// TIA Portal project "CropOne_SixRack" (V15.1)

(* hardware
DEVICE "ET 200SP station_1"  ET 200SP-Station
   slot 0: "Rack_0"  Rack  6ES5 710-8MAx1
   slot 1: "PLC"  CPU 1512SP-1 PN  6ES7 512-1DK01-0AB0  V2.6
   slot 2: "DQ 8x24VDC/0.5A ST_1"  DQ 8x24VDC/0.5A ST  6ES7 132-6BF01-0BA0  V0.0
      slot 1: "DQ 8x24VDC/0.5A ST_1"  DQ 8x24VDC/0.5A ST
   slot 3: "DQ 8x24VDC/0.5A ST_2"  DQ 8x24VDC/0.5A ST  6ES7 132-6BF01-0BA0  V0.0
      slot 1: "DQ 8x24VDC/0.5A ST_2"  DQ 8x24VDC/0.5A ST
   slot 4: "DQ 8x24VDC/0.5A ST_3"  DQ 8x24VDC/0.5A ST  6ES7 132-6BF01-0BA0  V0.0
      slot 1: "DQ 8x24VDC/0.5A ST_3"  DQ 8x24VDC/0.5A ST
   slot 5: "DQ 8x24VDC/0.5A ST_4"  DQ 8x24VDC/0.5A ST  6ES7 132-6BF01-0BA0  V0.0
      slot 1: "DQ 8x24VDC/0.5A ST_4"  DQ 8x24VDC/0.5A ST
   slot 6: "DQ 8x24VDC/0.5A ST_5"  DQ 8x24VDC/0.5A ST  6ES7 132-6BF01-0BA0  V0.0
      slot 1: "DQ 8x24VDC/0.5A ST_5"  DQ 8x24VDC/0.5A ST
   slot 7: "AI 4xU/I 2-wire ST_1"  AI 4xU/I 2-wire ST  6ES7 134-6HD01-0BA1  V2.0
      slot 1: "AI 4xU/I 2-wire ST_1"  AI 4xU/I 2-wire ST
   slot 8: "AI 4xU/I 2-wire ST_2"  AI 4xU/I 2-wire ST  6ES7 134-6HD01-0BA1  V2.0
      slot 1: "AI 4xU/I 2-wire ST_2"  AI 4xU/I 2-wire ST
   slot 9: "AI 4xU/I 2-wire ST_3"  AI 4xU/I 2-wire ST  6ES7 134-6HD01-0BA1  V2.0
      slot 1: "AI 4xU/I 2-wire ST_3"  AI 4xU/I 2-wire ST
   slot 10: "AI 4xU/I 2-wire ST_4"  AI 4xU/I 2-wire ST  6ES7 134-6HD01-0BA1  V2.0
      slot 1: "AI 4xU/I 2-wire ST_4"  AI 4xU/I 2-wire ST
   slot 11: "AI 4xU/I 2-wire ST_5"  AI 4xU/I 2-wire ST  6ES7 134-6HD01-0BA1  V2.0
      slot 1: "AI 4xU/I 2-wire ST_5"  AI 4xU/I 2-wire ST
   slot 12: "Server module_1"  Server module  6ES7 193-6PA00-0AA0  V1.1
      slot 1: "Server module_1"  Server module
   slot 127: "BA 2xRJ45"  BA 2xRJ45  6ES7 193-6AR00-0AA0  V0.0
      slot 32769: "Port_1"  6ES7 193-6AR00-0AA0
      slot 32770: "Port_2"  6ES7 193-6AR00-0AA0
DEVICE "SCALANCE S-600"  SCALANCE S-Station
   slot 0: "Rack"  Rail
   slot 0: "Router"  SCALANCE S615  6GK5 615-0AA00-2AA2  V5.0
DEVICE "SINAMICS G_1"  Sinamics.Device
   slot 0: "	_0"  Rail  SinamicsG120PRackP
   slot 0: "RackPumpVFD_1"  G120P CU230P-2 PN  6SL3243-0BB30-1FA0  4.7.10
      slot 1: "PROFINET interface"  MDD-SinamicsG120-P
   slot 3: "PM240-2 IP20"  PM240-2 IP20  6SL3210-1PB17-4ULx  -
DEVICE "ET 200SP station_2"  ET 200SP-Station
   slot 0: "Rack_0"  Rack  6ES5 710-8MAx1
   slot 0: "IO_Room_2"  IM 155-6 PN ST  6ES7 155-6AU01-0BN0  V4.1
   slot 1: "DQ 8x24VDC/0.5A ST_1"  DQ 8x24VDC/0.5A ST  6ES7 132-6BF01-0BA0  V0.0
      slot 1: "DQ 8x24VDC/0.5A ST_1"  DQ 8x24VDC/0.5A ST
   slot 2: "DQ 8x24VDC/0.5A ST_2"  DQ 8x24VDC/0.5A ST  6ES7 132-6BF01-0BA0  V0.0
      slot 1: "DQ 8x24VDC/0.5A ST_2"  DQ 8x24VDC/0.5A ST
   slot 3: "DQ 8x24VDC/0.5A ST_3"  DQ 8x24VDC/0.5A ST  6ES7 132-6BF01-0BA0  V0.0
      slot 1: "DQ 8x24VDC/0.5A ST_3"  DQ 8x24VDC/0.5A ST
   slot 4: "DQ 8x24VDC/0.5A ST_4"  DQ 8x24VDC/0.5A ST  6ES7 132-6BF01-0BA0  V0.0
      slot 1: "DQ 8x24VDC/0.5A ST_4"  DQ 8x24VDC/0.5A ST
   slot 5: "DQ 8x24VDC/0.5A ST_5"  DQ 8x24VDC/0.5A ST  6ES7 132-6BF01-0BA0  V0.0
      slot 1: "DQ 8x24VDC/0.5A ST_5"  DQ 8x24VDC/0.5A ST
   slot 6: "DQ 8x24VDC/0.5A ST_6"  DQ 8x24VDC/0.5A ST  6ES7 132-6BF00-0BA0  V1.1
      slot 1: "DQ 8x24VDC/0.5A ST_6"  DQ 8x24VDC/0.5A ST
   slot 7: "AI 4xU/I 2-wire ST_1"  AI 4xU/I 2-wire ST  6ES7 134-6HD01-0BA1  V2.0
      slot 1: "AI 4xU/I 2-wire ST_1"  AI 4xU/I 2-wire ST
   slot 8: "AI 4xU/I 2-wire ST_2"  AI 4xU/I 2-wire ST  6ES7 134-6HD01-0BA1  V2.0
      slot 1: "AI 4xU/I 2-wire ST_2"  AI 4xU/I 2-wire ST
   slot 9: "AI 4xU/I 2-wire ST_3"  AI 4xU/I 2-wire ST  6ES7 134-6HD01-0BA1  V2.0
      slot 1: "AI 4xU/I 2-wire ST_3"  AI 4xU/I 2-wire ST
   slot 10: "AI 4xU/I 2-wire ST_4"  AI 4xU/I 2-wire ST  6ES7 134-6HD01-0BA1  V2.0
      slot 1: "AI 4xU/I 2-wire ST_4"  AI 4xU/I 2-wire ST
   slot 11: "AI 4xU/I 2-wire ST_5"  AI 4xU/I 2-wire ST  6ES7 134-6HD01-0BA1  V2.0
      slot 1: "AI 4xU/I 2-wire ST_5"  AI 4xU/I 2-wire ST
   slot 12: "Server module_1"  Server module  6ES7 193-6PA00-0AA0  V1.1
      slot 1: "Server module_1"  Server module
   slot 127: "BA 2xRJ45"  BA 2xRJ45  6ES7 193-6AR00-0AA0  V0.0
      slot 1: "Port_1"  X1 P1 R  6ES7 193-6AR00-0AA0  V0.0
      slot 2: "Port_2"  X1 P2 R  6ES7 193-6AR00-0AA0  V0.0
DEVICE "HVAC_Modbus_1"  Dummy PC
   slot 1: "PROFINET interface"  PN-IO
DEVICE "HVAC_Modbus_2"  Dummy PC
   slot 1: "PROFINET interface"  PN-IO
DEVICE "SINAMICS G_2"  Sinamics.Device
   slot 0: "	_0"  Rail  SinamicsG120PRackP
   slot 0: "RackPumpVFD_2"  G120P CU230P-2 PN  6SL3243-0BB30-1FA0  4.7.10
      slot 1: "PROFINET interface"  MDD-SinamicsG120-P
   slot 3: "PM240-2 IP20"  PM240-2 IP20  6SL3210-1PB17-4ULx  -
DEVICE "SINAMICS G_3"  Sinamics.Device
   slot 0: "	_0"  Rail  SinamicsG120PRackP
   slot 0: "RackPumpVFD_3"  G120P CU230P-2 PN  6SL3243-0BB30-1FA0  4.7.10
      slot 1: "PROFINET interface"  MDD-SinamicsG120-P
   slot 3: "PM240-2 IP20"  PM240-2 IP20  6SL3210-1PB17-4ULx  -
DEVICE "SINAMICS G_4"  Sinamics.Device
   slot 0: "	_0"  Rail  SinamicsG120PRackP
   slot 0: "RackPumpVFD_4"  G120P CU230P-2 PN  6SL3243-0BB30-1FA0  4.7.10
      slot 1: "PROFINET interface"  MDD-SinamicsG120-P
   slot 3: "PM240-2 IP20"  PM240-2 IP20  6SL3210-1PB17-4ULx  -
DEVICE "SINAMICS G_5"  Sinamics.Device
   slot 0: "	_0"  Rail  SinamicsG120PRackP
   slot 0: "RackPumpVFD_5"  G120P CU230P-2 PN  6SL3243-0BB30-1FA0  4.7.10
      slot 1: "PROFINET interface"  MDD-SinamicsG120-P
   slot 3: "PM240-2 IP20"  PM240-2 IP20  6SL3210-1PB17-4ULx  -
DEVICE "SINAMICS G_6"  Sinamics.Device
   slot 0: "	_0"  Rail  SinamicsG120PRackP
   slot 0: "RackPumpVFD_6"  G120P CU230P-2 PN  6SL3243-0BB30-1FA0  4.7.10
      slot 1: "PROFINET interface"  MDD-SinamicsG120-P
   slot 3: "PM240-2 IP20"  PM240-2 IP20  6SL3210-1PB17-4ULx  -
*)

// ===== PLC "PLC"  CPU 1512SP-1 PN =====

VAR_GLOBAL CONSTANT   // PLC tag table "Library Constants"
   "eSTATE_MANUAL" : Int := 2;   // State Machine enumeration
   "ePBLT_FLASHING_ENABLED" : Int := 4;   // HMI PB LT enumeration
   "eSTATE_RETRACTING" : Int := 5;   // State Machine enumeration
   "IoScaling.S7Analog.Ni100.rScaledMax" : Real := 250.0;
   "IoScaling.S7Analog.Ni100.Climate.rScaledMax" : Real := 250.0;
   "eSTEP_StoppingStart" : Int := 4000;   // State Machine enumeration
   "eSTEP_VerifyCenterComplete" : Int := 7999;   // State Machine enumeration
   "IoScaling.S7Analog.150Ohms.rScaledMax" : Real := 150.0;
   "IoScaling.S7Analog.Default.bSwapBytes" : Bool := false;
   "eANALOG_INPUTHIGHHIGH" : Int := 102;
   "eMOTION_DISABLED" : Int := 4;   // Status Enumeration - Motion
   "IoScaling.S7Analog.Pt100.iRawMax" : Int := 8500;
   "eSTEP_RetractingComplete" : Int := 5999;   // State Machine enumeration
   "eMODE_MANUAL" : Int := 2;   // Mode enumeration
   "eANALOG_INPUTINVALID" : Int := 101;
   "ePBLT_HIDDEN" : Int := -1;   // HMI PB LT enumeration
   "eVALVE_HOMEON" : Int := 6;
   "IoScaling.S7Analog.Pt100.Climate.rScaledMin" : Real := -120.0;
   "eHOME_ABS_RET_ABS" : Int := 7;   // See MC_Home help for details
   "eMOTION_ERROR" : Int := 0;   // Status Enumeration - Motion
   "ePB_MAINTAINED" : Int := 1;   // HMI PB Type enumeration
   "LKINCTRL_LENGTH_OF_PATHDATA_NAME" : Int := 10;
   "LKINCTRL_NO_OF_PATHDATA_ELEMENTS" : Int := 15;
   "IoScaling.S7Analog.Pt100.Climate.iRawMax" : Int := 13000;
   "eVALVE_ERROR" : Int := 2;
   "IoScaling.S7Analog.Types.Pt100.Climate" : Int := 3;
   "eMODE_INDEPENDENT" : Int := 10;   // Mode
   "IoScaling.S7Analog.600Ohms.rScaledMax" : Real := 600.0;
   "eMOTION_RUNNING" : Int := 2;   // Status Enumeration - Motion
   "IoScaling.S7Analog.Ni100.Climate.rScaledMin" : Real := -60.0;
   "eMOTION_STOPPED" : Int := 1;   // Status Enumeration - Motion
   "eMOTION_MAINTENANCE" : Int := 3;   // Status Enumeration - Motion
   "IoScaling.S7Analog.Ni100.rScaledMin" : Real := -60.0;
   "eSTATE_STOPPING" : Int := 4;   // State Machine enumeration
   "IoScaling.S7Analog.Pt100.Climate.rScaledMax" : Real := 130.0;
   "IoScaling.S7Analog.Pt100.rScaledMax" : Real := 850.0;
   "IoScaling.S7Analog.Types.Ni100.Climate" : Int := 5;
   "ePB_UNLATCH" : Int := 3;   // HMI PB Type enumeration
   "IoScaling.S7Analog.Ni100.Climate.iRawMax" : Int := 25000;
   "eSTEP_BladeChangeStart" : Int := 6000;   // State Machine enumeration
   "IoScaling.S7Analog.300Ohms.rScaledMin" : Real := 0.0;
   "IoScaling.S7Analog.Types.Pt100" : Int := 2;
   "LKINCTRL_PI" : LReal := 3.1415926535897932846264;
   "eVALVE_WORKPOSITION" : Int := 3;
   "eCAM_SYNCDIRECTION_SHORTESTWAY" : Int := 3;   // See MC_CamIn help for details
   "IoScaling.S7Analog.Types.+-V/mA" : Int := 1;
   "ePBLT_FLASHING_DISABLED" : Int := 5;   // HMI PB LT enumeration
   "IoScaling.S7Analog.150Ohms.rScaledMin" : Real := 0.0;
   "eHOME_ACCEPT_CURRENT" : Int := 11;   // Used when the configured and current encoders don't match
   "LKINCTRL_NO_OF_START_EXECUTE_CMDS" : Int := 5;
   "ePBLT_TRANSITIONING" : Int := 2;   // HMI PB LT enumeration
   "SM_ACTIVE_DYNAMICS" : Int := 0;
   "eVALVE_WORKON" : Int := 5;
   "IoScaling.S7Analog.+-V/mA.iRawMax" : Int := 27648;
   "eSTATE_INITIALIZATION" : Int := 1;   // State Machine enumeration
   "LKINCTRL_NO_OF_PATHDATA_PREBUFFER_ELEMENTS" : Int := 5;
   "eHOME_ABS_RET_OFFSET" : Int := 6;   // See MC_Home help for details
   "eSTEP_BladeChangeComplete" : Int := 6999;   // State Machine enumeration
   "eSTEP_RunningComplete" : Int := 3999;   // State Machine enumeration
   "eANALOG_READY" : Int := 100;
   "ePBLT_ENABLED" : Int := 1;   // HMI PB LT enumeration
   "IoScaling.S7Analog.Pt100.Climate.iRawMin" : Int := -12000;
   "eSTATE_RUNNING" : Int := 3;   // State Machine enumeration
   "LKINCTRL_NO_OF_LAST_FLAG" : Int := 15;
   "IoScaling.S7Analog.Ni100.iRawMax" : Int := 2500;
   "IoScaling.S7Analog.Types.Default" : Int := 0;
   "eHOME_ACCEPT_CONFIG" : Int := 12;   // Used when the configured and current encoders don't match
   "eSTEP_RunningStart" : Int := 3000;   // State Machine enumeration
   "IoScaling.S7Analog.Default.iRawMin" : Int := 0;
   "ePBLT_ACTIVE" : Int := 3;   // HMI PB LT enumeration
   "IoScaling.S7Analog.Types.Ni100" : Int := 4;
   "eMODE_AUTO" : Int := 1;   // Mode enumeration
   "IoScaling.S7Analog.Default.iRawMax" : Int := 27648;
   "ePBLT_DISABLED" : Int := 0;   // HMI PB LT enumeration
   "LKINCTRL_NO_OF_SEQ_EXECUTE_CMDS" : Int := 5;
   "eSTEP_StoppingComplete" : Int := 4999;   // State Machine enumeration
   "IoScaling.S7Analog.Ni100.Climate.iRawMin" : Int := -6000;
   "IoScaling.S7Analog.Pt100.iRawMin" : Int := -2000;
   "ePB_LATCH" : Int := 2;   // HMI PB Type enumeration
   "eVALVE_ESTOP" : Int := 1;
   "eSTEP_RetractingStart" : Int := 5000;   // State Machine enumeration
   "IoScaling.S7Analog.300Ohms.rScaledMax" : Real := 300.0;
   "eANALOG_INPUTLOW" : Int := 105;
   "IoScaling.S7Analog.Pt100.rScaledMin" : Real := -200.0;
   "eSTATE_BLADECHANGE" : Int := 6;   // State Machine enumeration
   "IoScaling.S7Analog.600Ohms.rScaledMin" : Real := 0.0;
   "eSTATE_VERIFYCENTER" : Int := 7;   // State Machine enumeration
   "eVALVE_STOPPED" : Int := 0;
   "eCAM_SYNCPROFILEREFERENCE_LEADINGVALUEDISTANCE" : Int := 1;   // See MC_CamIn help for details
   "IoScaling.S7Analog.Ni100.iRawMin" : Int := -600;
   "ePB_HELD" : Int := 4;   // HMI PB Type enumeration
   "LKINCTRL_NO_OF_CMD_SETFLAGS" : Int := 8;
   "eSTEP_VerifyCenterStart" : Int := 7000;   // State Machine enumeration
   "eVALVE_HOMEPOSITION" : Int := 4;
   "eANALOG_INPUTHIGH" : Int := 104;
   "eANALOG_INPUTLOWLOW" : Int := 103;
   "IoScaling.S7Analog.+-V/mA.iRawMin" : Int := -27648;
   "ePB_MOMENTARY" : Int := 0;   // HMI PB Type enumeration
   "Modes.PID.Pretuning" : Int := 1;
   "TotalizerTimeUnits.DAYS" : Int := 4;
   "HMI.Status.ForwardWork" : Int := 3;
   "FIFO.iQueueDisabled" : Int := -1;
   "Handshakes.iSize" : Int := 5;
   "Modes.Auto" : Int := 1;
   "HMI.Status.Generic1" : Int := 101;
   "Simocode.Types.DirectStarter" : Int := 1;
   "Estop.MinSetPoint" : Int := 0;
   "Simocode.Types.OverloadRelay" : Int := 0;
   "HMI.Status.SimulatedReverseHome" : Int := 8;
   "TotalizerTimeUnits.MILLISECONDS" : Int := 0;
   "HMI.Status.Generic4" : Int := 104;
   "SoftStarter.HMI.Status.EStop" : Int := 1;
   "HMI.Status.OnForwardWork" : Int := 5;
   "DataTypes.iMaxInt" : Int := 32767;
   "FIFO.iQueueSize" : Int := 5;
   "Modes.PID.ManualMode" : Int := 4;
   "TotalizerTimeUnits.SECONDS" : Int := 1;
   "SoftStarter.Types.3RW30" : Int := 30;
   "HMI.Status.Generic3" : Int := 103;
   "HMI.Status.OnReverseHome" : Int := 6;
   "HMI.Status.Estop" : Int := 1;
   "SoftStarter.HMI.Status.Error" : Int := 2;
   "HMI.Status.Generic6" : Int := 106;
   "DataTypes.rMaxReal" : Real := 3.402823e38;
   "SoftStarter.HMI.Status.Off" : Int := 0;
   "Modes.PID.Inactive" : Int := 0;
   "HMI.Status.GenericNone" : Int := 100;
   "HMI.Status.Generic2" : Int := 102;
   "Modes.PID.AutoMode" : Int := 3;
   "SoftStarter.HMI.Status.On" : Int := 4;
   "Estop.HMISetPoint" : Int := 2;
   "HMI.Status.ReverseHome" : Int := 4;
   "DataTypes.rMinReal" : Real := -3.402823e38;
   "TotalizerTimeUnits.MINUTES" : Int := 2;
   "Modes.PID.FineTuning" : Int := 2;
   "TotalizerTimeUnits.HOURS" : Int := 3;
   "Ramp.Timed" : Int := 1;
   "Estop.MaxSetPoint" : Int := 1;
   "SoftStarter.Types.3RW40" : Int := 40;
   "Ramp.Continuous" : Int := 0;
   "HMI.Status.Generic5" : Int := 105;
   "Modes.Manual" : Int := 2;
   "Modes.Stop" : Int := 0;
   "HMI.Status.SimulatedOnReverseHome" : Int := 10;
   "Simocode.Types.ReversingStarter" : Int := 2;
   "Modes.Independent" : Int := 10;
   "DataTypes.iMinInt" : Int := -32768;
   "SoftStarter.HMI.Status.RampUp" : Int := 3;
   "SoftStarter.HMI.Status.RampDown" : Int := 5;
   "HMI.Status.Error" : Int := 2;
   "HMI.Status.SimulatedOnForwardWork" : Int := 9;
   "HMI.Status.SimulatedForwardWork" : Int := 7;
   "HMI.Status.Stopped" : Int := 0;
END_VAR

VAR_GLOBAL   // PLC tag table "IO"
   "GlobalAI" AT %I100.0 : "udtArrAIGlobal";
   "GlobalDQ" AT %Q100.0 : "udtArrDQGlobal";
END_VAR

VAR_GLOBAL CONSTANT   // PLC tag table "GLOBAL_CONSTANTS"
   "NUM_AI_RACK" : UInt := 1;   // Number of physical analog input points used per rack.
   "NUM_DQ_RACK" : UInt := 4;   // Number of physical digital output points used per rack.
   "NUM_DQ_ROOM" : UInt := 8;   // Number of physical digital output points used per room.
   "MAX_DQ_PER_ROOM" : UInt := 40;   // Max number of physical digital output points per room-based IO module. This needs to equal (NUM_DQ_ROOM + NUM_DQ_RACK*MAX_RACKS_PER_ROOM + EXTRA_DQ_PER_ROOM).
   "MAX_VFDS" : UInt := 6;   // Total number of VFDs configured in the HW config. This needs to equal MAX_ROOMS * MAX_RACKS_PER_ROOM.
   "MAX_ROOMS" : UInt := 1;   // Maximum possible number of rooms controlled by a given PLC
   "MAX_RACKS_PER_ROOM" : UInt := 6;   // Maximum possible number of racks per room
   "NUM_AI_ROOM" : UInt := 12;   // Number of physical analog input points used per room.
   "EXTRA_DQ_PER_ROOM" : UInt := 8;   // Number of unused physical digital output points per room-based IO module.
   "EXTRA_AI_PER_ROOM" : UInt := 2;   // Number of unused physical analog input points per room-based IO module.
   "MAX_AI_PER_ROOM" : UInt := 20;   // Max number of physical analog input points per room-based IO module. This needs to equal (NUM_AI_ROOM + NUM_AI_RACK*MAX_RACKS_PER_ROOM + EXTRA_AI_PER_ROOM).
END_VAR

VAR_GLOBAL   // PLC tag table "System Bits"
   "System_Byte" AT %MB1 : Byte;
   "AlwaysFALSE" AT %M1.3 : Bool;
   "Clock_1.25Hz" AT %M0.4 : Bool;
   "Clock_1Hz" AT %M0.5 : Bool;
   "Clock_0.5Hz" AT %M0.7 : Bool;
   "FirstScan" AT %M1.0 : Bool;
   "Clock_Byte" AT %MB0 : Byte;
   "Clock_2.5Hz" AT %M0.2 : Bool;
   "Clock_0.625Hz" AT %M0.6 : Bool;
   "Clock_5Hz" AT %M0.1 : Bool;
   "Clock_10Hz" AT %M0.0 : Bool;
   "AlwaysTRUE" AT %M1.2 : Bool;
   "DiagStatusUpdate" AT %M1.1 : Bool;
   "Clock_2Hz" AT %M0.3 : Bool;
END_VAR

VAR_GLOBAL   // PLC tag table "Temporary I/O"
   "Q_DischargeSolenoid" AT %Q0.2 : Bool;
   "Q_Rack3Supply" AT %Q1.5 : Bool;
   "Q_Rack4Lights" AT %Q3.4 : Bool;
   "IW_pHSensor" AT %IW12 : Int;
   "IW_RoomTemperature_1" AT %IW0 : Int;
   "Q_Rack6Supply" AT %Q2.6 : Bool;
   "Q_Rack5Lights" AT %Q3.5 : Bool;
   "Q_Rack4Supply" AT %Q2.0 : Bool;
   "Q_Rack1Return" AT %Q1.0 : Bool;
   "Q_Rack2Lights" AT %Q3.2 : Bool;
   "IW_NutrientALevel" AT %IW6 : Int;
   "Q_Rack3Lights" AT %Q3.3 : Bool;
   "Q_Rack2Shelves" AT %Q1.4 : Bool;
   "Q_FreshWaterSolenoid" AT %Q0.1 : Bool;
   "IW_Rack4Level" AT %IW24 : Int;
   "Q_MPathSolenoid" AT %Q0.0 : Bool;
   "Q_Rack4Shelves" AT %Q2.2 : Bool;
   "Q_Rack5Supply" AT %Q2.3 : Bool;
   "Q_NutrientAEnable" AT %Q0.4 : Bool;
   "IW_TankLevel" AT %IW4 : Int;
   "Q_Rack1Lights" AT %Q3.1 : Bool;
   "Q_Rack4Return" AT %Q2.1 : Bool;
   "Q_Rack6Lights" AT %Q3.6 : Bool;
   "IW_ISESensor" AT %IW16 : Int;
   "Q_Rack3Return" AT %Q1.6 : Bool;
   "Q_Rack6Shelves" AT %Q3.0 : Bool;
   "IW_NutrientAcidLevel" AT %IW10 : Int;
   "Q_Rack1Supply" AT %Q0.7 : Bool;
   "Q_NutrientMixingPumps" AT %Q3.7 : Bool;
   "Q_NutrientBEnable" AT %Q0.5 : Bool;
   "Q_Rack5Return" AT %Q2.4 : Bool;
   "Q_NutrientAcidEnable" AT %Q0.6 : Bool;
   "Q_Rack3Shelves" AT %Q1.7 : Bool;
   "Q_Rack2Return" AT %Q1.3 : Bool;
   "Q_Rack5Shelves" AT %Q2.5 : Bool;
   "IW_Rack2Level" AT %IW20 : Int;
   "IW_Rack6Level" AT %IW28 : Int;
   "IW_NutrientBLevel" AT %IW8 : Int;
   "Q_Rack1Shelves" AT %Q1.1 : Bool;
   "Q_Rack2Supply" AT %Q1.2 : Bool;
   "IW_Rack1Level" AT %IW18 : Int;
   "IW_RoomHumidity_1" AT %IW2 : Int;
   "IW_Rack3Level" AT %IW22 : Int;
   "Q_TankReturnSolenoid" AT %Q0.3 : Bool;
   "IW_Rack5Level" AT %IW26 : Int;
   "Q_Rack6Return" AT %Q2.7 : Bool;
   "IW_ECSensor" AT %IW14 : Int;
   "IW_RoomTemperature_2" AT %IW32 : Int;
   "IW_RoomHumidity_2" AT %IW34 : Int;
   "IW_ORPSensor" AT %IW36 : Int;
END_VAR

TYPE "udtTimeOfDaySetpoint"
   STRUCT
      TimeOfDaySeconds : DInt := -1;   // -1 default for unused setpoint
      rSetpoint : Real;
   END_STRUCT;
END_TYPE

TYPE "udtModbusValReal"
   STRUCT
      iRegister : UInt;   // Full modbus address (1 indexed, including offset for object type)
      rVal : Real;
   END_STRUCT;
END_TYPE

TYPE "udtNutrientReading"
   STRUCT
      rISEReading : Real;   // Nutrient measurement level
      rORPReading : Real;   // Nutrient measurement level
      rECReading : Real;   // Nutrient measurement level
      rpHReading : Real;   // Nutrient measurement level
   END_STRUCT;
END_TYPE

TYPE "udtModbusValBool"
   STRUCT
      iAddr : UInt;   // Full modbus address (1 indexed, including offset for object type)
      bVal : Bool;
   END_STRUCT;
END_TYPE

TYPE "udtFertigationSettings"
   STRUCT
      tMeasurementTime : Time;   // Duration of cycle through M loop before measurement taken (s)
      rMeasurementVolume : Real;   // Amount of water to receive from rack for measurement (L)
      bNutrientAEnable : Bool;   // Enables nutrient A for use in dosing
      bNutrientBEnable : Bool;   // Enables nutrient B for use in dosing
      rISELowSP : Real;   // Low setpoint for ISE measurement for dosing
      rISEHighSP : Real;   // High setpoint for ISE measurement for dosing
      tNutrientDosingDuration : Time;   // Duration for which to add a nutrient during dosing (s)
      bDosingActive : Bool;   // Rack was dosed on last MD cycle and is below high SP
      rOperatingVolume : Real;   // Operating volume for fill after dosing (L)
      rTotalShelfVolume : Real;
      rMaxReservoirVolume : Real;   // Maximum water capacity of the rack (L)
      rRackCurrentVolume : Real;   // Current rack fill level (L)
      bPumpAtStandstill : Bool;
      bEndDischargeCommand : Bool;
      tDischargeTime : Time;
      bEnableIncomingRotate : Bool;   // Rack is in M&D mode and circulating state
   END_STRUCT;
END_TYPE

// folder: IO

TYPE "udtDigitalOutput"
   STRUCT
      bAutoVal : Bool;   // Value set by the program
      bOverrideVal : Bool;   // Value set by the user, tracks bAuto when bOverrideEnable=0
      bStatus : Bool;   // Value being written to actual output
      bOverrideEnable : Bool;   // Sets bOut to bOverride
   END_STRUCT;
END_TYPE

TYPE "udtArrDQRoom"
   STRUCT
      DQ : Array[1.."MAX_DQ_PER_ROOM"] of Bool;
   END_STRUCT;
END_TYPE

TYPE "udtArrAIRoom"
   STRUCT
      AI : Array[1.."MAX_AI_PER_ROOM"] of Int;
   END_STRUCT;
END_TYPE

TYPE "udtArrDQGlobal"
   STRUCT
      Room : Array[1.."MAX_ROOMS"] of "udtArrDQRoom";
   END_STRUCT;
END_TYPE

TYPE "udtArrAIGlobal"
   STRUCT
      Room : Array[1.."MAX_ROOMS"] of "udtArrAIRoom";
   END_STRUCT;
END_TYPE

TYPE "udtRackDQ"
   STRUCT
      Q_SupplySolenoid : Bool;
      Q_ReturnSolenoid : Bool;
      Q_ShelfSolenoid : Bool;
      Q_Lights : Bool;
   END_STRUCT;
END_TYPE

TYPE "udtRoomAI"
   STRUCT
      IW_RoomTemperature_1 : Int;
      IW_RoomTemperature_2 : Int;
      IW_RoomHumidity_1 : Int;
      IW_RoomHumidity_2 : Int;
      IW_TankLevel : Int;
      IW_NutrientALevel : Int;
      IW_NutrientBLevel : Int;
      IW_NutrientAcidLevel : Int;
      IW_pHSensor : Int;
      IW_ECSensor : Int;
      IW_ISESensor : Int;
      IW_ORPSensor : Int;
   END_STRUCT;
END_TYPE

TYPE "udtRoomDQ"
   STRUCT
      Q_MPathSolenoid : Bool;
      Q_FreshWaterSolenoid : Bool;
      Q_DischargeSolenoid : Bool;
      Q_TankReturnSolenoid : Bool;
      Q_NutrientAEnable : Bool;
      Q_NutrientBEnable : Bool;
      Q_NutrientAcidEnable : Bool;
      Q_NutrientMixingPumps : Bool;
   END_STRUCT;
END_TYPE

TYPE "udtRackAI"
   STRUCT
      IW_ReservoirLevel : Int;
   END_STRUCT;
END_TYPE

// folder: Library Data Types/Error

TYPE "udtError_VFD"
VERSION : 0.1
   STRUCT
      MotorProtectorTripped : Bool;   // Motor protector tripped
      LocalDisconnectOff : Bool;   // Motor disconnect off
      ClutchTripped : Bool;   // Clutch tripped
      NoContactorFeedback : Bool;   // No feedback from motor contactor
      ContactorStillOn : Bool;   // Contactor still on
      NoSignalForward : Bool;   // No signal forward from VFD
      NoSignalReverse : Bool;   // No signal reverse from VFD
      MotorNotStopped : Bool;   // Motor doesn't stop
      MaxFrequencyReached : Bool;   // Max frequency reached
      Overcurrent : Bool;   // VFD overcurrent
      MotorOverload : Bool;   // Motor overload
      VFDOverload : Bool;   // VFD overload
      GeneralFault : Bool;   // VFD fault
      NoCoolingFanFeedback : Bool;   // No feedback from cooling fan
   END_STRUCT;
END_TYPE

// folder: Library Data Types/HMI

TYPE "udtHMI_VFD_Control"
VERSION : 0.1
   STRUCT
      iMode : Int;   // Current mode
      iErrorCode : Int;   // Error code
      iStatus : Int;   // Status for HMI display
      rManualSpeedSP : Real;   // Speed set point for manual mode
      rAutoSpeedSP : Real;   // Speed set point for automatic mode
      rActualSpeed : Real;   // Actual motor speed
      rActualCurrent : Real;   // Actual motor current
      rActualPower : Real;   // Actual motor power
      bPB_ResetError : Bool;   // PB Reset errors
      bPB_Forward : Bool;   // PB Move forward in manual mode
      bPB_Reverse : Bool;   // PB Move reverse in manual mode
      bPB_Stop : Bool;   // PB Stop in manual mode
      bPBEN_ResetError : Bool;   // PB Reset errors enabled
      bPBEN_Forward : Bool;   // PB Forward enabled
      bPBEN_Reverse : Bool;   // PB Reverse enabled
      bPBEN_Stop : Bool;   // PB Stop enabled
      bForwardOn : Bool;   // Moving forward
      bReverseOn : Bool;   // Moving Reverse
      bSignalForward : Bool;   // Forward signal
      bSignalReverse : Bool;   // Reverse signal
      bError : Bool;   // Overall error
      bInterlock : Bool;   // VFD Interlocked
   END_STRUCT;
END_TYPE

// folder: (top level)

DATA_BLOCK "dbMain"   // DB6
{ S7_Optimized_Access := 'TRUE' }
VERSION : 0.1
// stored: InstanceOfName fbMain
"fbMain"
BEGIN
END_DATA_BLOCK

FUNCTION_BLOCK "fbRoomHVAC"   // FB2, LAD
{ S7_Optimized_Access := 'TRUE' }
VERSION : 0.1
   VAR
      Temperature_Cooling : "fbAlarmedSetpoint";
      Humidity : "fbAlarmedSetpoint";
      CO2 : "fbAlarmedSetpoint";
   END_VAR
   VAR RETAIN
      Controls : Struct
         rHeatingSP : Real := 55.0;
         bResetAlarm : Bool;
         bResetModbus : Bool;
      END_STRUCT;
   END_VAR
   VAR
      Status : Struct
         rSupplyAirTemperature : Real;
         bModbusError : Bool;
         wLastModbusErrorCode : Word;
         Compressor_1_Percentage : Real;
         Compressor_2_Percentage : Real;
         ZoneAirEnthalpy : Real;
         Compressor_1_Command : Bool;
         Compressor_1_Enabled : Bool;
         Compressor_1_Alarm : Bool;
         Compressor_2_Command : Bool;
         Compressor_2_Enabled : Bool;
         Compressor_2_Alarm : Bool;
         LPS1_Alarm : Bool;
         LPS2_Alarm : Bool;
         HPS1_Alarm : Bool;
         HPS2_Alarm : Bool;
      END_STRUCT;
   END_VAR
   VAR RETAIN
      Config : Struct
         ModbusServerAddr : IP_V4;   // IP address for Modbus TCP server
         ID : UInt := 81;   // Unique ID for connection, also used as port number on PLC
      END_STRUCT;
   END_VAR
   VAR
      TCPConnection : TCON_IP_v4;
      fbModbusTCPClient_Instance : "fbModbusTCPClient";
      Read_Discrete : Array[0..9] of "udtModbusValBool";
      Write_Discrete : Array[0..0] of "udtModbusValBool";
      Read_Registers : Array[0..6] of "udtModbusValReal";
      Write_Registers : Array[0..2] of "udtModbusValReal";
   END_VAR
   VAR CONSTANT
      cFakeScaling : Int := 150;
      cRoomTempIndex : Int := 0;
      cHumidityIndex : Int := 1;
      cCO2Index : Int := 2;
      cSupplyAirTempIndex : Int := 3;
   END_VAR
   // TCPConnection.RemotePort := 502;
   // TCPConnection.ActiveEstablished := true;
   // TCPConnection.ConnectionType := 11;
   // Config.ModbusServerAddr.ADDR[2] := 1;
   // Config.ModbusServerAddr.ADDR[1] := 10;
   // TCPConnection.LocalPort := 1001;
   // TCPConnection.RemoteAddress.ADDR[1] := 10;
   // TCPConnection.RemoteAddress.ADDR[2] := 1;
   // TCPConnection.RemoteAddress.ADDR[3] := 0;
   // TCPConnection.RemoteAddress.ADDR[4] := 20;
   // Config.ModbusServerAddr.ADDR[3] := 0;
   // Config.ModbusServerAddr.ADDR[4] := 20;
   // Temperature_Cooling.arrSetpoints[1].rSetpoint := 75.0;
   // Humidity.arrSetpoints[1].rSetpoint := 55.0;
BEGIN

REGION Network 1 (SCL): Set connection parameters
   #TCPConnection.InterfaceId := "Local~PROFINET_interface_1"; // PLC ethernet port
   #TCPConnection.ID := UINT_TO_WORD(#Config.ID);
   #TCPConnection.ConnectionType := 11; // TCP
   #TCPConnection.ActiveEstablished := TRUE;
   #TCPConnection.RemoteAddress := #Config.ModbusServerAddr;
   #TCPConnection.RemotePort := 502; // Default for Modbus TCP
   #TCPConnection.LocalPort := #Config.ID;
END_REGION

REGION Network 2 (SCL): Set up registers
   // Read coils and discrete inputs (00001 and 10001)
   #Read_Discrete[0].iAddr := 10048; // Compressor_1_Command
   #Read_Discrete[1].iAddr := 10067; // Compressor_1_Enabled
   #Read_Discrete[2].iAddr := 10091; // Compressor_1_Alarm
   #Read_Discrete[3].iAddr := 10049; // Compressor_2_Command
   #Read_Discrete[4].iAddr := 10008; // Compressor_2_Enabled
   #Read_Discrete[5].iAddr := 10068; // Compressor_2_Alarm
   #Read_Discrete[6].iAddr := 10089; // LPS1_Alarm
   #Read_Discrete[7].iAddr := 10034; // LPS2_Alarm
   #Read_Discrete[8].iAddr := 10093; // HPS1_Alarm
   #Read_Discrete[9].iAddr := 10097; // HPS2_Alarm

   // Write coils (00001)
   #Write_Discrete[0].iAddr := 00020; // Alarm reset
   #Write_Discrete[0].bVal := #Controls.bResetAlarm;

   // Read input and holding registers (30001 and 40001)
   #Read_Registers[#cRoomTempIndex].iRegister      := 30035; // Room Temperature
   #Read_Registers[#cHumidityIndex].iRegister      := 30031; // Humidity
   #Read_Registers[#cCO2Index].iRegister           := 30001; // CO2
   #Read_Registers[#cSupplyAirTempIndex].iRegister := 30043; // Supply Air Temperature

   #Read_Registers[4].iRegister := 30077; // Compressor_1_percentage
   #Read_Registers[5].iRegister := 30049; // Compressor_2_percentage
   #Read_Registers[6].iRegister := 30039; // ZoneAirEnthalpy

   // Write holding registers (40001)
   #Write_Registers[0].iRegister := 40119; // Cooling SP
   #Write_Registers[0].rVal := #Temperature_Cooling.rSetpoint;

   #Write_Registers[1].iRegister := 40121; // Heating SP
   #Write_Registers[1].rVal := #Controls.rHeatingSP;

   #Write_Registers[2].iRegister := 40097; // Dehumidification SP
   #Write_Registers[2].rVal := #Humidity.rSetpoint;
   (*
   #Write_Data[3].iRegister := 2; // CO2 SP 1
   #Write_Data[3].rVal := #CO2.rSetpoint;

   #Write_Data[4].iRegister := 66; // CO2 SP 2
   #Write_Data[4].rVal := #CO2.rSetpoint;
   *)
END_REGION

REGION Network 3: Modbus TCP Client Block Call
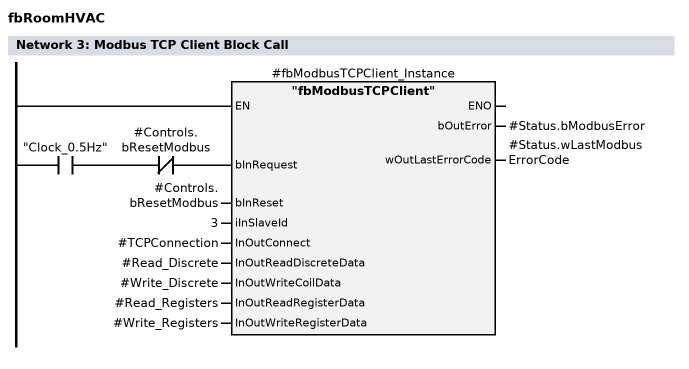
   RUNG wire#powerrail
      #fbModbusTCPClient_Instance(bInRequest := wire#w1, bInReset := #Controls.bResetModbus, iInSlaveId := 3, InOutConnect := #TCPConnection, InOutReadDiscreteData := #Read_Discrete, InOutWriteCoilData := #Write_Discrete, InOutReadRegisterData := #Read_Registers, InOutWriteRegisterData := #Write_Registers, bOutError => #Status.bModbusError, wOutLastErrorCode => #Status.wLastModbusErrorCode)
   END_RUNG
   RUNG wire#powerrail
      Contact( "Clock_0.5Hz" )
      I_Contact( #Controls.bResetModbus )
   END_RUNG wire#w1
   // the same network as SCL:
   #fbModbusTCPClient_Instance(bInRequest := "Clock_0.5Hz" AND NOT #Controls.bResetModbus,   // "fbModbusTCPClient"
                           bInReset := #Controls.bResetModbus,
                           iInSlaveId := 3,
                           InOutConnect := #TCPConnection,
                           InOutReadDiscreteData := #Read_Discrete,
                           InOutWriteCoilData := #Write_Discrete,
                           InOutReadRegisterData := #Read_Registers,
                           InOutWriteRegisterData := #Write_Registers,
                           bOutError => #Status.bModbusError,
                           wOutLastErrorCode => #Status.wLastModbusErrorCode);
END_REGION

REGION Network 4 (SCL): Parse received data
   // Status data
   #Status.Compressor_1_Percentage := #Read_Registers[4].rVal;
   #Status.Compressor_2_Percentage := #Read_Registers[5].rVal;
   #Status.ZoneAirEnthalpy := #Read_Registers[6].rVal;

   #Status.Compressor_1_Command := #Read_Discrete[0].bVal;
   #Status.Compressor_1_Enabled := #Read_Discrete[1].bVal;
   #Status.Compressor_1_Alarm :=   #Read_Discrete[2].bVal;
   #Status.Compressor_2_Command := #Read_Discrete[3].bVal;
   #Status.Compressor_2_Enabled := #Read_Discrete[4].bVal;
   #Status.Compressor_2_Alarm :=   #Read_Discrete[5].bVal;
   #Status.LPS1_Alarm := #Read_Discrete[6].bVal;
   #Status.LPS2_Alarm := #Read_Discrete[7].bVal;
   #Status.HPS1_Alarm := #Read_Discrete[8].bVal;
   #Status.HPS2_Alarm := #Read_Discrete[9].bVal;


   // Bypass analog scaling for alarmed setpoints
   #Temperature_Cooling.Config.rLowCalibration := 0;
   #Temperature_Cooling.Config.rHighCalibration := #cFakeScaling;
   #Humidity.Config.rLowCalibration := 0;
   #Humidity.Config.rHighCalibration := #cFakeScaling;
   #CO2.Config.rLowCalibration := 0;
   #CO2.Config.rHighCalibration := #cFakeScaling;

   #Temperature_Cooling(
                        iInRawValue := REAL_TO_INT(#Read_Registers[#cRoomTempIndex].rVal /
                                                   #cFakeScaling * "IoScaling.S7Analog.Default.iRawMax"));

   #Humidity(
             iInRawValue := REAL_TO_INT(#Read_Registers[#cHumidityIndex].rVal /
                                        #cFakeScaling * "IoScaling.S7Analog.Default.iRawMax"));

   #CO2(
        iInRawValue := REAL_TO_INT(#Read_Registers[#cCO2Index].rVal /
                                   #cFakeScaling * "IoScaling.S7Analog.Default.iRawMax"));

   #Status.rSupplyAirTemperature := #Read_Registers[#cSupplyAirTempIndex].rVal;
END_REGION
END_FUNCTION_BLOCK

FUNCTION_BLOCK "fbRoom"   // FB3, LAD
{ S7_Optimized_Access := 'TRUE' }
VERSION : 0.1
   VAR_INPUT
      arrAI : Array[1.."NUM_AI_ROOM"] of Int;
      AI AT arrAI : "udtRoomAI";
   END_VAR
   VAR_OUTPUT
      arrDQ : Array[1.."NUM_DQ_ROOM"] of Bool;
      DQ AT arrDQ : "udtRoomDQ";
   END_VAR
   VAR
      Rack : Array[1.."MAX_RACKS_PER_ROOM"] of "fbRack";
      Fertigation : "fbRoomFertigation";
      HVAC : "fbRoomHVAC";
   END_VAR
   VAR RETAIN
      Config : Struct
         iNumRacks : Int := 1;
      END_STRUCT;
   END_VAR
   VAR
      AI_Temperature_1 : "fbAlarmedSetpoint";
      AI_Temperature_2 : "fbAlarmedSetpoint";
      AI_Humidity_1 : "fbAlarmedSetpoint";
      AI_Humidity_2 : "fbAlarmedSetpoint";
      AI_TankLevel : "fbAlarmedSetpoint";
      AI_NutrientALevel : "fbAlarmedSetpoint";
      AI_NutrientBLevel : "fbAlarmedSetpoint";
      AI_NutrientAcidLevel : "fbAlarmedSetpoint";
      AI_pHSensor : "fbAlarmedSetpoint";
      AI_ECSensor : "fbAlarmedSetpoint";
      AI_ISESensor : "fbAlarmedSetpoint";
      AI_ORPSensor : "fbAlarmedSetpoint";
   END_VAR
   VAR RETAIN
      DQ_MPathSolenoid : "udtDigitalOutput";
      DQ_FreshWaterSolenoid : "udtDigitalOutput";
      DQ_DischargeSolenoid : "udtDigitalOutput";
      DQ_TankReturnSolenoid : "udtDigitalOutput";
      DQ_NutrientA : "udtDigitalOutput";
      DQ_NutrientB : "udtDigitalOutput";
      DQ_NutrientAcid : "udtDigitalOutput";
      DQ_NutrientMixing : "udtDigitalOutput";
   END_VAR
   VAR
      arrFertigationSettings : Array[0.."MAX_RACKS_PER_ROOM"] of "udtFertigationSettings";
   END_VAR
   VAR_TEMP
      i : Int;   // Index for iterating through racks
   END_VAR
   // AI_NutrientALevel.Config.rLowCalibration := 0.0;
   // AI_NutrientALevel.Config.rHighCalibration := 200.0;
   // AI_NutrientBLevel.Config.rLowCalibration := 0.0;
   // AI_NutrientBLevel.Config.rHighCalibration := 200.0;
   // AI_NutrientAcidLevel.Config.rLowCalibration := 0.0;
   // AI_NutrientAcidLevel.Config.rHighCalibration := 200.0;
   // AI_TankLevel.Config.rLowCalibration := 0.0;
   // AI_TankLevel.Config.rHighCalibration := 1085.0;
   // AI_Temperature_1.Config.rLowCalibration := -40.0;
   // AI_Temperature_1.Config.rHighCalibration := 140.0;
   // AI_Temperature_2.Config.rLowCalibration := -40.0;
   // AI_Temperature_2.Config.rHighCalibration := 140.0;
   // AI_Humidity_1.Config.rLowCalibration := 0.0;
   // AI_Humidity_1.Config.rHighCalibration := 100.0;
   // AI_Humidity_2.Config.rLowCalibration := 0.0;
   // AI_Humidity_2.Config.rHighCalibration := 100.0;
   // AI_ORPSensor.Config.rLowCalibration := -1500.0;
   // AI_ORPSensor.Config.rHighCalibration := 1500.0;
   // AI_pHSensor.Config.rLowCalibration := 0.0;
   // AI_pHSensor.Config.rHighCalibration := 14.0;
   // AI_ECSensor.Config.rLowCalibration := 0.0;
   // AI_ECSensor.Config.rHighCalibration := 5.0;
   // AI_ISESensor.Config.rLowCalibration := 0.0;
   // AI_ISESensor.Config.rHighCalibration := 10000.0;
BEGIN

REGION Network 1 (SCL): Process room-level analog inputs
   #AI_Temperature_1(#AI.IW_RoomTemperature_1);
   #AI_Temperature_2(#AI.IW_RoomTemperature_2);
   #AI_Humidity_1(#AI.IW_RoomHumidity_1);
   #AI_Humidity_2(#AI.IW_RoomHumidity_2);
   #AI_TankLevel(#AI.IW_TankLevel);
   #AI_NutrientALevel(#AI.IW_NutrientALevel);
   #AI_NutrientBLevel(#AI.IW_NutrientBLevel);
   #AI_NutrientAcidLevel(#AI.IW_NutrientAcidLevel);
   #AI_pHSensor(#AI.IW_pHSensor);
   #AI_ECSensor(#AI.IW_ECSensor);
   #AI_ISESensor(#AI.IW_ISESensor);
   #AI_ORPSensor(#AI.IW_ORPSensor);
END_REGION

REGION Network 2 (SCL): Call rack FBs
   FOR #i := 1 TO #Config.iNumRacks DO

       #Rack[#i](iInMutexLockConfirmation := #Fertigation.arrOutMutexLocks[#i],
                 udtInLastNutrientReading := #Fertigation.arrOutNutrientReading[#i],
                 bInSupplySolenoidFromRoomFertigation := #Fertigation.arrOutSupplySolenoids[#i],
                 bInReturnSolenoidFromRoomFertigation := #Fertigation.arrOutReturnSolenoids[#i],
                 iInLightsDelaySecs := #i * 5000, // delay each rack by 5 seconds to prevent current spike
                 arrAI := #Rack[#i].arrAI,
                 iOutMutexRequest => #Fertigation.arrInMutexRequests[#i],
                 OutFertigationSettings => #arrFertigationSettings[#i],
                 arrDQ => #Rack[#i].arrDQ);
   END_FOR;
END_REGION

REGION Network 3 (SCL): Call room-level fertigation control logic and map rack supply and return solenoids
   #Fertigation(arrInMutexRequests:=#Fertigation.arrInMutexRequests,
                arrInFertigationSettings:=#arrFertigationSettings,
                rInTankLevel:=#AI_TankLevel.rActual,
                rInNutrientALevel:=#AI_NutrientALevel.rActual,
                rInNutrientBLevel:=#AI_NutrientBLevel.rActual,
                rInNutrientAcidLevel:=#AI_NutrientAcidLevel.rActual,
                rInpHSensor:=#AI_pHSensor.rActual,
                rInECSensor:=#AI_ECSensor.rActual,
                rInISESensor:=#AI_ISESensor.rActual,
                rInORPReading:=#AI_ORPSensor.rActual,
                iInNumRacks:=#Config.iNumRacks,
                bOutTankReturnSolenoid=>#Fertigation.bOutTankReturnSolenoid,
                bOutMPathSolenoid=>#Fertigation.bOutMPathSolenoid,
                bOutFreshWaterSolenoid=>#Fertigation.bOutFreshWaterSolenoid,
                bOutDischargeSolenoid=>#Fertigation.bOutDischargeSolenoid,
                bOutNutrientMixing=>#Fertigation.bOutNutrientMixing,
                bOutNutrientA=>#Fertigation.bOutNutrientA,
                bOutNutrientB=>#Fertigation.bOutNutrientB,
                bOutNutrientAcid=>#Fertigation.bOutNutrientAcid,
                arrOutNutrientReading=>#Fertigation.arrOutNutrientReading,
                arrOutMutexLocks=>#Fertigation.arrOutMutexLocks,
                arrOutSupplySolenoids=>#Fertigation.arrOutSupplySolenoids,
                arrOutReturnSolenoids=>#Fertigation.arrOutReturnSolenoids);
END_REGION

REGION Network 4 (SCL): Set room-level outputs
   #DQ.Q_MPathSolenoid := "fcDigitalOutput"(bInAutoVal := #Fertigation.bOutMPathSolenoid, InOutUdt := #DQ_MPathSolenoid);
   #DQ.Q_FreshWaterSolenoid := "fcDigitalOutput"(bInAutoVal := #Fertigation.bOutFreshWaterSolenoid, InOutUdt := #DQ_FreshWaterSolenoid);
   #DQ.Q_DischargeSolenoid := "fcDigitalOutput"(bInAutoVal := #Fertigation.#bOutDischargeSolenoid, InOutUdt := #DQ_DischargeSolenoid);
   #DQ.Q_TankReturnSolenoid := "fcDigitalOutput"(bInAutoVal := #Fertigation.bOutTankReturnSolenoid, InOutUdt := #DQ_TankReturnSolenoid);
   #DQ.Q_NutrientAEnable := "fcDigitalOutput"(bInAutoVal := #Fertigation.#bOutNutrientA, InOutUdt := #DQ_NutrientA);
   #DQ.Q_NutrientBEnable := "fcDigitalOutput"(bInAutoVal := #Fertigation.#bOutNutrientB, InOutUdt := #DQ_NutrientB);
   #DQ.Q_NutrientAcidEnable := "fcDigitalOutput"(bInAutoVal := #Fertigation.#bOutNutrientAcid, InOutUdt := #DQ_NutrientAcid);
   #DQ.Q_NutrientMixingPumps := "fcDigitalOutput"(bInAutoVal := #Fertigation.#bOutNutrientMixing, InOutUdt := #DQ_NutrientMixing);
END_REGION

REGION Network 5: Call HVAC FB
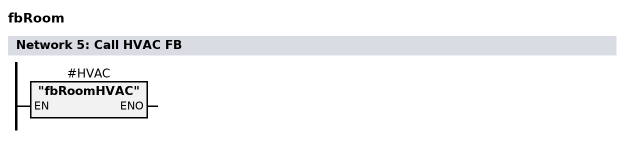
   RUNG wire#powerrail
      #HVAC()
   END_RUNG
   // the same network as SCL:
   #HVAC();   // "fbRoomHVAC"
END_REGION
END_FUNCTION_BLOCK

FUNCTION_BLOCK "fbMain"   // FB4, LAD
{ S7_Optimized_Access := 'TRUE' }
VERSION : 0.1
// Main block which calls all room FBs and holds all parameters in instance memory.
   VAR
      Room : Array[1.."MAX_ROOMS"] of "fbRoom";
      Config : "fbConfig";
   END_VAR
   VAR_TEMP
      iRoomCount : Int;
      iRackCount : Int;
      iPos : DInt;
   END_VAR
BEGIN

REGION Network 1 (SCL): Call config FB
   // bInSimulation := TRUE skips IO device configuration steps
   #Config(bInSimulation := #Config.bInSimulation);
END_REGION

REGION Network 2 (SCL): Map input array to all room and rack inputs
   IF #Config.Status.bDone THEN

       FOR #iRoomCount := 1 TO UINT_TO_INT("MAX_ROOMS") DO

           #iPos := 1; // input array is 1 indexed

           MOVE_BLK(IN := "GlobalAI".Room[#iRoomCount].AI[#iPos],
                    COUNT := "NUM_AI_ROOM",
                    OUT => #Room[#iRoomCount].arrAI[1]);

           #iPos += "NUM_AI_ROOM";


           FOR #iRackCount := 1 TO UINT_TO_INT("MAX_RACKS_PER_ROOM") DO

               MOVE_BLK(IN := "GlobalAI".Room[#iRoomCount].AI[#iPos],
                        COUNT := "NUM_AI_RACK",
                        OUT => #Room[#iRoomCount].Rack[#iRackCount].arrAI[1]);

               #iPos += "NUM_AI_RACK";

           END_FOR;

           #iPos += "EXTRA_AI_PER_ROOM"; // skip over unused points

       END_FOR;

   END_IF;
END_REGION

REGION Network 3 (SCL): TEMPORARY- Remap inputs from temporary IO tag table
   #Room[1].arrAI[1] := "IW_RoomTemperature_1";
   #Room[1].arrAI[2] := "IW_RoomTemperature_2";
   #Room[1].arrAI[3] := "IW_RoomHumidity_1";
   #Room[1].arrAI[4] := "IW_RoomHumidity_2";
   #Room[1].arrAI[5] := "IW_TankLevel";
   #Room[1].arrAI[6] := "IW_NutrientALevel";
   #Room[1].arrAI[7] := "IW_NutrientBLevel";
   #Room[1].arrAI[8] := "IW_NutrientAcidLevel";
   #Room[1].arrAI[9] := "IW_pHSensor";
   #Room[1].arrAI[10] := "IW_ECSensor";
   #Room[1].arrAI[11] := "IW_ISESensor";
   #Room[1].arrAI[12] := "IW_ORPSensor";

   #Room[1].Rack[1].arrAI[1] := "IW_Rack1Level";
   #Room[1].Rack[2].arrAI[1] := "IW_Rack2Level";
   #Room[1].Rack[3].arrAI[1] := "IW_Rack3Level";
   #Room[1].Rack[4].arrAI[1] := "IW_Rack4Level";
   #Room[1].Rack[5].arrAI[1] := "IW_Rack5Level";
   #Room[1].Rack[6].arrAI[1] := "IW_Rack6Level";
END_REGION

REGION Network 4 (SCL): Call FBs for all configured rooms
   IF #Config.Status.bDone THEN

       FOR #iRoomCount := 1 TO #Config.iNumRooms DO

           #Room[#iRoomCount](arrAI := #Room[#iRoomCount].arrAI,
                              arrDQ=> #Room[#iRoomCount].arrDQ);

       END_FOR;

   END_IF;
END_REGION

REGION Network 5 (SCL): Combine all room and rack outputs into a single output array
   IF #Config.Status.bDone THEN

       FOR #iRoomCount := 1 TO UINT_TO_INT("MAX_ROOMS") DO

           #iPos := 1; // output array is 1 indexed

           MOVE_BLK(IN := #Room[#iRoomCount].arrDQ[1],
                    COUNT := "NUM_DQ_ROOM",
                    OUT => "GlobalDQ".Room[#iRoomCount].DQ[#iPos]);

           #iPos += "NUM_DQ_ROOM";


           FOR #iRackCount := 1 TO UINT_TO_INT("MAX_RACKS_PER_ROOM") DO

               MOVE_BLK(IN := #Room[#iRoomCount].Rack[#iRackCount].arrDQ[1],
                        COUNT := "NUM_DQ_RACK",
                        OUT => "GlobalDQ".Room[#iRoomCount].DQ[#iPos]);

               #iPos += "NUM_DQ_RACK";

           END_FOR;

           #iPos += "EXTRA_DQ_PER_ROOM"; // skip over unused points

       END_FOR;

   END_IF;
END_REGION

REGION Network 6 (SCL): TEMPORARY- Remap inputs to temporary IO tag table
   "Q_MPathSolenoid" := #Room[1].arrDQ[1];
   "Q_FreshWaterSolenoid" := #Room[1].arrDQ[2];
   "Q_DischargeSolenoid" := #Room[1].arrDQ[3];
   "Q_TankReturnSolenoid" := #Room[1].arrDQ[4];
   "Q_NutrientAEnable" := #Room[1].arrDQ[5];
   "Q_NutrientBEnable" := #Room[1].arrDQ[6];
   "Q_NutrientAcidEnable" := #Room[1].arrDQ[7];
   "Q_NutrientMixingPumps" := #Room[1].arrDQ[8];

   "Q_Rack1Supply" := #Room[1].Rack[1].arrDQ[1];
   "Q_Rack1Return" := #Room[1].Rack[1].arrDQ[2];
   "Q_Rack1Shelves" := #Room[1].Rack[1].arrDQ[3];
   "Q_Rack1Lights" := #Room[1].Rack[1].arrDQ[4];
   "Q_Rack2Supply" := #Room[1].Rack[2].arrDQ[1];
   "Q_Rack2Return" := #Room[1].Rack[2].arrDQ[2];
   "Q_Rack2Shelves" := #Room[1].Rack[2].arrDQ[3];
   "Q_Rack2Lights" := #Room[1].Rack[2].arrDQ[4];
   "Q_Rack3Supply" := #Room[1].Rack[3].arrDQ[1];
   "Q_Rack3Return" := #Room[1].Rack[3].arrDQ[2];
   "Q_Rack3Shelves" := #Room[1].Rack[3].arrDQ[3];
   "Q_Rack3Lights" := #Room[1].Rack[3].arrDQ[4];
   "Q_Rack4Supply" := #Room[1].Rack[4].arrDQ[1];
   "Q_Rack4Return" := #Room[1].Rack[4].arrDQ[2];
   "Q_Rack4Shelves" := #Room[1].Rack[4].arrDQ[3];
   "Q_Rack4Lights" := #Room[1].Rack[4].arrDQ[4];
   "Q_Rack5Supply" := #Room[1].Rack[5].arrDQ[1];
   "Q_Rack5Return" := #Room[1].Rack[5].arrDQ[2];
   "Q_Rack5Shelves" := #Room[1].Rack[5].arrDQ[3];
   "Q_Rack5Lights" := #Room[1].Rack[5].arrDQ[4];
   "Q_Rack6Supply" := #Room[1].Rack[6].arrDQ[1];
   "Q_Rack6Return" := #Room[1].Rack[6].arrDQ[2];
   "Q_Rack6Shelves" := #Room[1].Rack[6].arrDQ[3];
   "Q_Rack6Lights" := #Room[1].Rack[6].arrDQ[4];
END_REGION
END_FUNCTION_BLOCK

FUNCTION_BLOCK "fbRack"   // FB5, LAD
{ S7_Optimized_Access := 'TRUE' }
VERSION : 0.1
   VAR_INPUT
      iInMutexLockConfirmation : Int;
      udtInLastNutrientReading : "udtNutrientReading";
      bInSupplySolenoidFromRoomFertigation : Bool;
      bInReturnSolenoidFromRoomFertigation : Bool;
      iInLightsDelaySecs : Int;
      arrAI : Array[1.."NUM_AI_RACK"] of Int;
      AI AT arrAI : "udtRackAI";
   END_VAR
   VAR_OUTPUT
      iOutMutexRequest : Int;
      OutFertigationSettings : "udtFertigationSettings";
      arrDQ : Array[1.."NUM_DQ_RACK"] of Bool;
      DQ AT arrDQ : "udtRackDQ";
   END_VAR
   VAR
      Lighting : "fbRackLights";
      Fertigation : "fbRackFertigation";
      AI_ReservoirLevel : "fbAlarmedSetpoint";
   END_VAR
   VAR RETAIN
      DQ_SupplySolenoid : "udtDigitalOutput";
      DQ_ReturnSolenoid : "udtDigitalOutput";
      DQ_ShelfSolenoid : "udtDigitalOutput";
      DQ_Lights : "udtDigitalOutput";
   END_VAR
   // AI_ReservoirLevel.Config.rLowCalibration := 0.0;
   // AI_ReservoirLevel.Config.rHighCalibration := 951.0;
BEGIN

REGION Network 1 (SCL)
   // Note that rack supply/return solenoids are managed by room-level fertigation FB
   // Process rack-level analog inputs
   #AI_ReservoirLevel(#AI.IW_ReservoirLevel);

   // Call lighting control fb
   #Lighting(iInDelaySecs:= #iInLightsDelaySecs,
             bOutLights => #Lighting.bOutLights);

   // Call rack-level fertigation logic
   #Fertigation(iInMutexLockConfirmation := #iInMutexLockConfirmation,
                InLastNutrientReading:= #udtInLastNutrientReading,
                rInReservoirLevel := #AI_ReservoirLevel.rActual,
                bInReturnSolenoidStatus:=#DQ.Q_ReturnSolenoid,
                bInShelfSolenoidStatus:=#DQ.Q_ShelfSolenoid,
                iOutMutexRequest => #iOutMutexRequest,
                OutFertigationSettings => #OutFertigationSettings,
                bOutShelfSolenoid => #Fertigation.bOutShelfSolenoid);

   // Set rack-level outputs
   // Rack supply/return solenoids are managed by room-level fertigation FB
   #DQ.Q_SupplySolenoid := "fcDigitalOutput"(bInAutoVal := #bInSupplySolenoidFromRoomFertigation, InOutUdt := #DQ_SupplySolenoid);
   #DQ.Q_ReturnSolenoid := "fcDigitalOutput"(bInAutoVal := #bInReturnSolenoidFromRoomFertigation, InOutUdt := #DQ_ReturnSolenoid);
   #DQ.Q_ShelfSolenoid  := "fcDigitalOutput"(bInAutoVal := #Fertigation.bOutShelfSolenoid, InOutUdt := #DQ_ShelfSolenoid);
   #DQ.Q_Lights         := "fcDigitalOutput"(bInAutoVal := #Lighting.bOutLights, InOutUdt := #DQ_Lights);
END_REGION
END_FUNCTION_BLOCK

FUNCTION_BLOCK "fbRackLights"   // FB6, LAD
{ S7_Optimized_Access := 'TRUE' }
VERSION : 0.1
   VAR_INPUT
      iInDelaySecs : Int;
   END_VAR
   VAR_OUTPUT
      bOutLights : Bool;
   END_VAR
   VAR RETAIN
      Controls : Struct
         iMode : Int;   // 0: Off, 1: On, 2: Auto
         diOffTime : DInt;   // Off time (seconds past midnight)
         diOnTime : DInt;   // On time (seconds past midnight)
      END_STRUCT;
   END_VAR
   VAR
      Status : Struct
         diSecondsElapsed : DInt;
      END_STRUCT;
      bLightsCommand : Bool;
      TON_OnDelay : TON_TIME;
   END_VAR
   VAR_TEMP
      tCurrentDateTime : Date_And_Time;   // Current PLC Date and Time
      tCurrentTimeMilli : Time_Of_Day;   // Current time (ms since 0:00:00)
      retVal : Int;   // Garbage return value from RD_LOC_T
      diSeconds : DInt;
   END_VAR
   VAR CONSTANT
      eOffMode : Int := 0;
      eOnMode : Int := 1;
      eAutoMode : Int := 2;
   END_VAR
BEGIN

REGION Network 1 (SCL): State 0 - Off Mode and State 1 - On Mode
   // Directly assign rack light output based on off or on mode
   IF #Controls.iMode = #eOffMode THEN
       #bLightsCommand := 0;
   ELSIF #Controls.iMode = #eOnMode THEN
       #bLightsCommand := 1;
   END_IF;
END_REGION

REGION Network 2 (SCL): State 2 - Auto Mode
   // Check the current time against the on time and off time, and assign the lights appropriately
   IF #Controls.iMode = #eAutoMode THEN

       //Get current time from PLC and convert to seconds since 0:00:00
       #retVal := RD_LOC_T(OUT => #tCurrentDateTime);
       #tCurrentTimeMilli := DT_TO_TOD(IN := #tCurrentDateTime);
       #diSeconds := TOD_TO_DINT(IN := #tCurrentTimeMilli)/1000; //Go from ms time to DInt seconds

       // Situation 1: Off time happens after on time
       IF #Controls.diOffTime > #Controls.diOnTime THEN 
           IF #diSeconds > #Controls.diOnTime AND #diSeconds < #Controls.diOffTime THEN
               #bLightsCommand := 1;
           ELSE
               #bLightsCommand := 0;
           END_IF;

       // Situation 2: On time happens after off time
       ELSE
           IF #diSeconds > #Controls.diOffTime AND #diSeconds < #Controls.diOnTime THEN
               #bLightsCommand := 0;
           ELSE
               #bLightsCommand := 1;
           END_IF;
       END_IF;
   END_IF;
END_REGION

REGION Network 3 (SCL): Write seconds elapsed status and set outputs with confugred delay
   #Status.diSecondsElapsed := #diSeconds;

   #TON_OnDelay(IN := #bLightsCommand,
                PT := INT_TO_TIME(#iInDelaySecs));

   #bOutLights := #TON_OnDelay.Q;
END_REGION
END_FUNCTION_BLOCK

FUNCTION_BLOCK "fbRackFertigation"   // FB7, SCL
{ S7_Optimized_Access := 'TRUE' }
VERSION : 0.1
   VAR_INPUT
      iInMutexLockConfirmation : Int;   // 0: Off, 1: Fill, 2: Measurement/Dosing, 3:Discharge
      InLastNutrientReading : "udtNutrientReading";
      rInReservoirLevel : Real;   // Rack reservoir level
      bInReturnSolenoidStatus : Bool;   // Return solenoid status for determining when return to main tank or discharge
      bInShelfSolenoidStatus : Bool;
   END_VAR
   VAR_OUTPUT
      iOutMutexRequest : Int;   // 0: Off, 1: Fill, 2: Measurement/Dosing, 3:Discharge
      OutFertigationSettings : "udtFertigationSettings";
      bOutShelfSolenoid : Bool;
   END_VAR
   VAR RETAIN
      Controls : Struct
         iModeCommand : Int;   // 0: Off, 1: Fill, 2: Measurement/Dosing, 3:Discharge, 4: Circulate
         bEndDischargeCommand : Bool;   // Command to end discharge before timer expires
         diDischargeTimeSecs : DInt := 3600;   // Discharge duration (seconds)
         rPumpReservoirInterlockLevel : Real := 180.0;   // Reservoir level below which to turn off pump (L)
         rPumpContinousSpeed : Real := 79.2;   // Commanded pump speed (%)
         rPumpReturnSpeed : Real := 80.8;   // Commanded pump speed (%)
         rPumpDischargeSpeed : Real := 91.7;   // Commanded pump speed (%)
         diMeasurementSecs : DInt := 600;   // Duration of measurement (seconds)
         diDosingIntervalMins : DInt := 120;   // Time to stay in circulate mode before trigerring a M&D routine
         rMeasurementVolume : Real := 200.0;   // Volume to move from reservoir to tank during measurement
         iISEModeCommand : Int := 1;   // 0: Off, 1: Load, 2: Deplete
         bNutrientAEnable : Bool := true;   // Enable nutrient A for dosing
         bNutrientBEnable : Bool := true;   // Enable nutrient B for dosing
         rISELowSP : Real := 35.0;   // Low ISE setpoint for dosing
         rISEHighSP : Real := 145.0;   // High ISE setpoint for dosing
         diNutrientDosingSecs : DInt := 60;   // Duration of nutrient dosing (seconds)
         rOperatingVolume : Real := 450.0;   // Operating volume for rack reservoir (L)
         rTotalShelfVolume : Real := 1800.0;   // Total volume of the shelves (L)
         rMaxReservoirVolume : Real := 900.0;   // Maximum water capacity of the rack reservoir (L)
      END_STRUCT;
      Status : Struct
         iState : Int;   // 0: Off, 1: Fill, 2: Measurement/Dosing, 3:Discharge, 4: Circulate
         NutrientLevels : "udtNutrientReading";   // Last measured nutrient levels
      END_STRUCT;
   END_VAR
   VAR
      Pump : "fbRackPump";
   END_VAR
   VAR RETAIN
      bShelfSolenoidCommand : Bool;   // Command for shelf solenoid
      bLockConfirmedModeActive : Bool;   // Memory bit for mutex lock, used to detect lock dropping out
      iNextMode : Int;   // Holder for next user commanded mode
      rInitialVolume : Real;   // Initial volume of reservoir at start of measurement
   END_VAR
   VAR
      NutrientReadingReady : F_TRIG;
      TON_Circulate : TON_TIME;
   END_VAR
   VAR_TEMP
      rPumpSpeed : Real;
   END_VAR
   VAR CONSTANT
      eRackMode_Off : Int := 0;   // Rack Off State
      eRackMode_Fill : Int := 1;   // Rack Fill State
      eRackMode_MeasurementDosing : Int := 2;   // Rack Measurement and Dosing State
      eRackMode_Discharge : Int := 3;   // Rack Discharge State
      eRackMode_Circulate : Int := 4;   // Rack Circulate State
      eISEMode_Off : Int := 0;   // Skip dosing for this rack
      eISEMode_Load : Int := 1;   // Dose nutrients up to ISE High SP
      eISEMode_Deplete : Int := 2;   // Does nutrients up to ISE Low SP
   END_VAR
BEGIN
   // Rack Level Fertigation Controller
   // Responsible for: sending mutex lock requests to room, managing shelf valve and rack pump, and controlling rack state
   // Rack States:
   //      0 - Off
   //      1 - Fill
   //      2 - Measurement and Dosing
   //      3 - Discharge
   //      4 - Circulate (Default State)




   REGION 0: Off
       // In the off state, close the shelf solenoid and turn off the pump
       IF #Status.iState = #eRackMode_Off  THEN
           #iOutMutexRequest := #eRackMode_Off;
       END_IF;

       // wait to turn off shelf solenoid until pump stops
       IF #Status.iState = #eRackMode_Off AND #Pump.Status.rActualSpeed = 0 THEN
           #bShelfSolenoidCommand := 0;
       END_IF;

   END_REGION

   REGION 1: Fill
       // In the fill state, send the mutex lock request, wait for confirmation, run the pump and open the shelf solenoid
       // once the mutex lock drops out, move directly to 4: Circulate and set commanded mode to Circulate

       IF #Status.iState = #eRackMode_Fill THEN

           IF (#iInMutexLockConfirmation <> #eRackMode_Fill) AND NOT #bLockConfirmedModeActive THEN
               #iOutMutexRequest := #eRackMode_Fill;
           ELSIF #iInMutexLockConfirmation = #eRackMode_Fill THEN
               #bLockConfirmedModeActive := 1;
               #iOutMutexRequest := #eRackMode_Off;
               #bShelfSolenoidCommand := 1;
           ELSIF (#iInMutexLockConfirmation <> #eRackMode_Fill) AND #bLockConfirmedModeActive THEN
               #bLockConfirmedModeActive := 0;
               #iNextMode := #eRackMode_Circulate;
               #Controls.iModeCommand := #eRackMode_Circulate;
           END_IF;
       END_IF;


   END_REGION

   REGION 2: Measurement & Dosing
       // In the measurement and dosing state, send the mutex lock request along with the nutrient
       // dosing setpoints, wait for confirmation, then automatically transition TO 4: Circulation

       IF #Status.iState = #eRackMode_MeasurementDosing THEN

           // request M&D lock
           IF (#iInMutexLockConfirmation <> #eRackMode_MeasurementDosing) AND NOT #bLockConfirmedModeActive THEN
               #iOutMutexRequest := #eRackMode_MeasurementDosing;

               // confirm that we are locked
           ELSIF #iInMutexLockConfirmation = #eRackMode_MeasurementDosing AND NOT #bLockConfirmedModeActive THEN
               #bLockConfirmedModeActive := 1;
               #iOutMutexRequest := #eRackMode_Off;
               #bShelfSolenoidCommand := 1;
               #rInitialVolume := #rInReservoirLevel;

               // check that M&D is done, go back to circulate
           ELSIF #iInMutexLockConfirmation <> #eRackMode_MeasurementDosing AND #bLockConfirmedModeActive THEN
               #bLockConfirmedModeActive := 0;
               #iNextMode := #eRackMode_Circulate;
           END_IF;

       END_IF;


   END_REGION

   REGION 3: Discharge
       // In the discharge state, send the mutex lock request, wait for confirmation, close shelf solenoid
       // once the mutex lock drops out, move directly to 0: Off and set commanded mode to Off

       IF #Status.iState = #eRackMode_Discharge THEN
           IF (#iInMutexLockConfirmation <> #eRackMode_Discharge) AND NOT #bLockConfirmedModeActive THEN
               #iOutMutexRequest := #eRackMode_Discharge;
           ELSIF #iInMutexLockConfirmation = #eRackMode_Discharge THEN
               #bLockConfirmedModeActive := 1;
               #iOutMutexRequest := #eRackMode_Off;
               #bShelfSolenoidCommand := 0;
           ELSIF (#iInMutexLockConfirmation <> #eRackMode_Discharge) AND #bLockConfirmedModeActive THEN
               #bLockConfirmedModeActive := 0;
               #iNextMode := #eRackMode_Off;
               #Controls.iModeCommand := #eRackMode_Off;
           END_IF;
       ELSE
           #Controls.bEndDischargeCommand := FALSE;
       END_IF;

       #OutFertigationSettings.tDischargeTime := DINT_TO_TIME(#Controls.diDischargeTimeSecs * 1000);
       #OutFertigationSettings.bEndDischargeCommand := #Controls.bEndDischargeCommand;

   END_REGION

   REGION 4: Circulate
       // In the circulate state, open the shelf solenoid and run the pump
       // Mutex request to Room is off
       IF #Status.iState = #eRackMode_Circulate THEN
           #bShelfSolenoidCommand := 1;
           #iOutMutexRequest := #eRackMode_Off;
       END_IF;

       // Automatically trigger M&D after 2 hours of circulating if the commanded state is M&D
       #TON_Circulate(IN := #Status.iState = #eRackMode_Circulate AND #Controls.iModeCommand = #eRackMode_MeasurementDosing,
                      PT := DINT_TO_TIME(#Controls.diDosingIntervalMins * 60 * 1000));

       IF #TON_Circulate.Q THEN
           #iNextMode := #eRackMode_MeasurementDosing;
       END_IF;

   END_REGION

   REGION State Management
       // If rack is in Off or Circulate, take the OPC commanded state
       // Except if commanding M&D, go into circulate first, then it will automatically go into M&D on the timer
       // If rack is in M&D, Fill, or Discharge, wait for the automatic state transition

       IF #Status.iState = #eRackMode_Off  AND #Controls.iModeCommand = #eRackMode_MeasurementDosing THEN
           #iNextMode := #eRackMode_Circulate;

       ELSIF #Status.iState = #eRackMode_Off OR 
           (#Status.iState = #eRackMode_Circulate AND #Controls.iModeCommand <> #eRackMode_MeasurementDosing) THEN
           #iNextMode := #Controls.iModeCommand;

       END_IF;

       #Status.iState := #iNextMode;

   END_REGION


   REGION Pump Management

       IF #rInReservoirLevel < #Controls.rPumpReservoirInterlockLevel OR #Status.iState = #eRackMode_Off THEN
           // turn off pump if there's not enough water
           #rPumpSpeed := 0;

       ELSIF #Status.iState = #eRackMode_MeasurementDosing AND #bInReturnSolenoidStatus = 1 THEN
           // returning water to the main tank, check that the return solenoid is open
           #rPumpSpeed := #Controls.rPumpReturnSpeed;

       ELSIF #Status.iState = #eRackMode_Discharge AND #bInReturnSolenoidStatus = 1 THEN
           // discharging water from rack reservoir to sewer, check that the return solenoid is open
           #rPumpSpeed := #Controls.rPumpDischargeSpeed;

       ELSIF  #bInShelfSolenoidStatus = 1 THEN
           // circulate mode, fill mode, and all other state, double check the the shelf solenoid is open
           #rPumpSpeed := #Controls.rPumpContinousSpeed;

       ELSE
           #rPumpSpeed := 0;

       END_IF;

       #Pump(rInSpeedCommand := #rPumpSpeed);

   END_REGION

   REGION Fertigation Settings
       // Package up OPC Settings for fertigation to pass out to room

       #OutFertigationSettings.tMeasurementTime := DINT_TO_TIME(#Controls.diMeasurementSecs * 1000);
       #OutFertigationSettings.rMeasurementVolume := #Controls.rMeasurementVolume;
       #OutFertigationSettings.bNutrientAEnable := #Controls.bNutrientAEnable;
       #OutFertigationSettings.bNutrientBEnable := #Controls.bNutrientBEnable;
       #OutFertigationSettings.rISELowSP := #Controls.rISELowSP;
       #OutFertigationSettings.rISEHighSP := #Controls.rISEHighSP;
       #OutFertigationSettings.tNutrientDosingDuration := DINT_TO_TIME(#Controls.diNutrientDosingSecs * 1000);

       #OutFertigationSettings.rOperatingVolume := #Controls.rOperatingVolume;
       #OutFertigationSettings.rTotalShelfVolume := #Controls.rTotalShelfVolume;
       #OutFertigationSettings.rMaxReservoirVolume := #Controls.rMaxReservoirVolume;
       #OutFertigationSettings.rRackCurrentVolume := #rInReservoirLevel;

       #OutFertigationSettings.bPumpAtStandstill := #Pump.Status.rActualSpeed = 0;

       // Enable incoming rotate from room if in M&D mode and current state is circulate
       #OutFertigationSettings.bEnableIncomingRotate := #Status.iState = #eRackMode_Circulate
                                                         AND #Controls.iModeCommand = #eRackMode_MeasurementDosing;

       REGION ISE Mode
           // Determine if dosing is required based off of ISE reading, low/high setpoints, and commanded ISE mode

           // if in load mode and high SP is reached, switch to deplete
           IF #Controls.iISEModeCommand = #eISEMode_Load AND #InLastNutrientReading.rISEReading >= #Controls.rISEHighSP THEN
               #Controls.iISEModeCommand := #eISEMode_Deplete;
           END_IF;

           // if in deplete mode and low SP is reached, switch to load
           IF #Controls.iISEModeCommand = #eISEMode_Deplete AND #InLastNutrientReading.rISEReading <= #Controls.rISELowSP THEN
               #Controls.iISEModeCommand := #eISEMode_Load;
           END_IF;

           // Request dosing if in load mode, skip dosing if in deplete or off
           #OutFertigationSettings.bDosingActive := (#Controls.iISEModeCommand = #eISEMode_Load);

       END_REGION

       //Copy over nutrient levels to OPC status output when M&D lock drops out
       #NutrientReadingReady(CLK:= (#iInMutexLockConfirmation = #eRackMode_MeasurementDosing));
       IF #NutrientReadingReady.Q THEN
           #Status.NutrientLevels := #InLastNutrientReading;
       END_IF;


   END_REGION

   REGION Set digital outputs
       #bOutShelfSolenoid :=  #bShelfSolenoidCommand;

   END_REGION
END_FUNCTION_BLOCK

FUNCTION_BLOCK "fbRoomFertigation"   // FB8, SCL
{ S7_Optimized_Access := 'TRUE' }
VERSION : 0.1
   VAR_INPUT
      arrInMutexRequests : Array[0.."MAX_RACKS_PER_ROOM"] of Int;   // Array of mutex requests from racks
      arrInFertigationSettings : Array[0.."MAX_RACKS_PER_ROOM"] of "udtFertigationSettings";
      rInTankLevel : Real;
      rInNutrientALevel : Real;
      rInNutrientBLevel : Real;
      rInNutrientAcidLevel : Real;
      rInpHSensor : Real;
      rInECSensor : Real;
      rInISESensor : Real;
      rInORPReading : Real;
      iInNumRacks : Int;   // Number of racks to process mutex requests for
   END_VAR
   VAR_OUTPUT
      bOutTankReturnSolenoid : Bool;
      bOutMPathSolenoid : Bool;
      bOutFreshWaterSolenoid : Bool;
      bOutDischargeSolenoid : Bool;
      bOutNutrientMixing : Bool;
      bOutNutrientA : Bool;
      bOutNutrientB : Bool;
      bOutNutrientAcid : Bool;
      arrOutNutrientReading : Array[0.."MAX_RACKS_PER_ROOM"] of "udtNutrientReading";   // Array of nutrient readings going to racks
      arrOutMutexLocks : Array[0.."MAX_RACKS_PER_ROOM"] of Int;   // Array of mutex locks going to racks
      arrOutSupplySolenoids : Array[0.."MAX_RACKS_PER_ROOM"] of Bool;   // Array of supply solenoids for each rack
      arrOutReturnSolenoids : Array[0.."MAX_RACKS_PER_ROOM"] of Bool;   // Array of return solenoids for each rack
   END_VAR
   VAR RETAIN
      Controls : Struct
         bPauseFertigation : Bool;   // While true, prevents next rack from locking
         rFloorPumpSpeedSP : Real;   // Floor pump speed (RPM)
         iNutrientMixingMode : Int;   // Nutrient mixing mode (0: off, 1: on, 2: 10 minute, 3: Continuous)
         rFreshLevelForMeasurementLoop : Real;   // Amount of fresh water to fill in the tank during rotate to clean measurement loop
         rFillLevelToPreviousShelf : Real := 8.0;   // Amount of water to push back to previous tank during return
         rReturnPathVolume : Real := 19.0;   // Return path volume (L) to fill from active rack
         rTankEmptyLevel : Real := 150.0;   // Volume at which tank is considered empty (L)
         rTankMaxVolume : Real := 900.0;   // Maximum volume for tank (L)
      END_STRUCT;
   END_VAR
   VAR
      Status : Struct
         iState : Int;   // Current operation (0: off, 1: Fill, 2:Measurement/Dosing, 3:Discharge)
         iActiveRack : Int;   // Rack that currently has a lock, 0 if idle
         iLastMDRack : Int;   // Keep track of previous rack for rotate and flush, 0 if previous operation was not measurement and dosing
      END_STRUCT;
      bTankReturnSolenoidCommand : Bool;   // Command for tank return solenoid
      bMPathSolenoidCommand : Bool;   // Command for measurement path solenoid
      bFreshWaterSolenoidCommand : Bool;   // Command for fresh water solenoid
      bDischargeSolenoidCommand : Bool;   // Command for discharge solenoid
      bNutrientMixingCommand : Bool;   // Command for nutrient mixing enable
      bNutrientACommand : Bool;   // Command for dosing nutrient A
      bNutrientBCommand : Bool;   // Command for dosing nutrient B
      bNutrientAcidCommand : Bool;
      TON_Discharge : TON_TIME;
      TON_24HourNutrientMix : TON_TIME;
      fbRoomMeasurementDosing : "fbRoomMeasurementDosing";
      bTransferring : Bool;   // Memory bit for transfer to rack during fill process
      rTransferredVolume : Real;
      rVolumeToTransfer : Real;
      bEndDischarge : Bool;
   END_VAR
   VAR_TEMP
      bFoundActive : Bool;
      i : Int;   // Iterable for mutex request
      tCurrentDateTime : Date_And_Time;   // Current PLC Date and Time
      tCurrentTime : Time_Of_Day;   // Current PLC Time of Day
      retVal : Int;   // Garbage return value from RD_LOC_T
      bMDDone : Bool;
      rTargetFillVolume : Real;
   END_VAR
   VAR CONSTANT
      eRoomMode_Off : Int := 0;   // Room Off State
      eRoomMode_Fill : Int := 1;   // Room Filling State
      eRoomMode_MeasurementDosing : Int := 2;   // Room Measurement and Dosing State
      eRoomMode_Discharge : Int := 3;   // Room Discharge State
      eNutrientMixingMode_Off : Int := 0;   // Forced off
      eNutrientMixingMode_On : Int := 1;   // Forced on
      eNutrientMixingMode_TenMinute : Int := 2;   // Run for 10 minutes at noon
      eNutrientMixingMode_FullDay : Int := 3;   // Run for 24 hours then switch to Ten Minute mode
      MIX_START_TIME : Time_Of_Day := TOD#12:00:00;   // Start of 10 minute mix at noon
      MIX_END_TIME : Time_Of_Day := TOD#12:10:00;   // End of 10 minute mix at noon
   END_VAR
BEGIN
   REGION 0: Off
       // Close all solenoids
       // Iterate through mutex requests to trigger state change
       // Send lock when mutex request arrives

       IF #Status.iState = #eRoomMode_Off THEN
           #bTankReturnSolenoidCommand := 0;
           #bMPathSolenoidCommand := 0;
           #bFreshWaterSolenoidCommand := 0;

           IF NOT #Controls.bPauseFertigation THEN // if not paused, check for next rack requesting lock
               #bFoundActive := 0;
               FOR #i := 1 TO #iInNumRacks DO
                   IF #arrInMutexRequests[#i] <> #eRoomMode_Off THEN

                       // Mutex request active - update state and active rack, send lock
                       #Status.iState := #arrInMutexRequests[#i];
                       #Status.iActiveRack := #i;
                       #arrOutMutexLocks[#i] := #Status.iState;
                       #bFoundActive := 1;
                       //Break out of for loop
                       EXIT;
                   END_IF;
               END_FOR;
               IF NOT #bFoundActive THEN
                   #Status.iActiveRack := 0;
               END_IF; 
           END_IF;
       END_IF;


   END_REGION

   REGION 1: Fill
       // Open fresh water solenoid, fill until max volume reached or rack volume reached, close fresh water solenoid
       // Open rack supply solenoid, activate floor pump, wait for main tank content to return to rack

       // Need to keep track of how much has been sent to the rack, until total volume added matches OperatingVolume + TotalShelfVolume or
       // resevoir reaches max volume

       IF #Status.iState = #eRoomMode_Fill THEN

           #Status.iLastMDRack := 0; // no rotate if last rack last rack was filled

           #rTargetFillVolume := #arrInFertigationSettings[#Status.iActiveRack].rOperatingVolume
           + #arrInFertigationSettings[#Status.iActiveRack].rTotalShelfVolume;

           IF #rTransferredVolume >= #rTargetFillVolume OR
               #arrInFertigationSettings[#Status.iActiveRack].rRackCurrentVolume > #arrInFertigationSettings[#Status.iActiveRack].rMaxReservoirVolume THEN
               // Full volume or rack reservoir is too full, done with fill
               #Status.iState := #eRoomMode_Off;
               #arrOutMutexLocks[#Status.iActiveRack] := 0;

               #arrOutSupplySolenoids[#Status.iActiveRack] := 0;
               #bFreshWaterSolenoidCommand := 0;

               #bTransferring := 0;
               #rTransferredVolume := 0;


           ELSIF #rInTankLevel < #Controls.rTankMaxVolume AND
               #rInTankLevel - #Controls.rTankEmptyLevel + #rTransferredVolume < #rTargetFillVolume AND
               NOT #bTransferring THEN
               // Adding water to the main tank
               #bFreshWaterSolenoidCommand := 1;

           ELSIF NOT #bTransferring THEN
               // Start transfer from main tank to rack
               #bTransferring := 1;
               #bFreshWaterSolenoidCommand := 0;
               #rVolumeToTransfer := #rInTankLevel - #Controls.rTankEmptyLevel;

           END_IF;

           IF #bTransferring AND #rInTankLevel <= #Controls.rTankEmptyLevel THEN
               // Transfer is done, add volume to transferred total
               #bTransferring := 0;
               #rTransferredVolume += #rVolumeToTransfer;
               #rVolumeToTransfer := 0;
               #arrOutSupplySolenoids[#Status.iActiveRack] := 0;

           END_IF;

           // Transfer from main tank to rack until main tank is empty
           #arrOutSupplySolenoids[#Status.iActiveRack] := #bTransferring;

       END_IF;


   END_REGION


   REGION 2: Measurement AND Dosing
       // Call measurement and dosing subfunction for the room
       // Only write to outputs when in the correct mode

       // Reset the last rack id to skip rotate if that rack is not accepting rotate
       IF #Status.iState = #eRoomMode_MeasurementDosing AND #Status.iLastMDRack <> 0 THEN
           IF NOT #arrInFertigationSettings[#Status.iLastMDRack].bEnableIncomingRotate THEN
               #Status.iLastMDRack := 0;
           END_IF;
       END_IF;

        #fbRoomMeasurementDosing(bInStart := (#Status.iState = #eRoomMode_MeasurementDosing),
                                 iInActiveRack := #Status.iActiveRack,
                                 iInPreviousRack := #Status.iLastMDRack,
                                 rInTankLevel := #rInTankLevel,
                                 rInRackLevel := #arrInFertigationSettings[#Status.iActiveRack].rRackCurrentVolume,
                                 rInISEReading := #rInISESensor,
                                 rInECReading := #rInECSensor,
                                 rInpHReading := #rInpHSensor,
                                 rInORPReading := #rInORPReading,
                                 rInFillLevelToPreviousShelf := #Controls.rFillLevelToPreviousShelf,
                                 rInFreshLevelForMLoop := #Controls.rFreshLevelForMeasurementLoop,
                                 rInReturnPathVolume := #Controls.rReturnPathVolume,
                                 rInTankEmptyLevel := #Controls.rTankEmptyLevel,
                                 InFertigationSettings := #arrInFertigationSettings[#Status.iActiveRack],
                                 bOutTankReturnSolenoidCommand => #fbRoomMeasurementDosing.bOutTankReturnSolenoidCommand,
                                 bOutActiveRackReturnSolenoidCommand => #fbRoomMeasurementDosing.bOutActiveRackReturnSolenoidCommand,
                                 bOutActiveRackSupplySolenoidCommand => #fbRoomMeasurementDosing.bOutActiveRackSupplySolenoidCommand,
                                 bOutPreviousRackReturnSolenoidCommand => #fbRoomMeasurementDosing.bOutPreviousRackReturnSolenoidCommand,
                                 bOutPreviousRackSupplySolenoidCommand => #fbRoomMeasurementDosing.bOutPreviousRackSupplySolenoidCommand,
                                 bOutFreshWaterSolenoidCommand => #fbRoomMeasurementDosing.bOutFreshWaterSolenoidCommand,
                                 bOutDischargeSolenoidCommand => #fbRoomMeasurementDosing.bOutDischargeSolenoidCommand,
                                 bOutMPathSolenoidCommand => #fbRoomMeasurementDosing.bOutMPathSolenoidCommand,
                                 bOutNutrientACommand => #fbRoomMeasurementDosing.bOutNutrientACommand,
                                 bOutNutrientBCommand => #fbRoomMeasurementDosing.bOutNutrientBCommand,
                                 OutNutrientReadings => #fbRoomMeasurementDosing.OutNutrientReadings,
                                 bOutDone => #bMDDone);

       //Handle output writing
       IF #Status.iState = #eRoomMode_MeasurementDosing THEN
           #bTankReturnSolenoidCommand := #fbRoomMeasurementDosing.bOutTankReturnSolenoidCommand;
           #bFreshWaterSolenoidCommand := #fbRoomMeasurementDosing.bOutFreshWaterSolenoidCommand;
           #bDischargeSolenoidCommand := #fbRoomMeasurementDosing.bOutDischargeSolenoidCommand;
           #bMPathSolenoidCommand := #fbRoomMeasurementDosing.bOutMPathSolenoidCommand;
           #bNutrientACommand := #fbRoomMeasurementDosing.bOutNutrientACommand;
           #bNutrientBCommand := #fbRoomMeasurementDosing.bOutNutrientBCommand;
           #arrOutReturnSolenoids[#Status.iActiveRack] := #fbRoomMeasurementDosing.bOutActiveRackReturnSolenoidCommand;
           #arrOutSupplySolenoids[#Status.iActiveRack] := #fbRoomMeasurementDosing.bOutActiveRackSupplySolenoidCommand;
           #arrOutReturnSolenoids[#Status.iLastMDRack] := #fbRoomMeasurementDosing.bOutPreviousRackReturnSolenoidCommand;
           #arrOutSupplySolenoids[#Status.iLastMDRack] := #fbRoomMeasurementDosing.bOutPreviousRackSupplySolenoidCommand;
           #arrOutNutrientReading[#Status.iActiveRack] := #fbRoomMeasurementDosing.OutNutrientReadings;

           IF #bMDDone THEN
               #Status.iState := #eRoomMode_Off;
               #arrOutMutexLocks[#Status.iActiveRack] := #eRoomMode_Off;
               #Status.iLastMDRack := #Status.iActiveRack; // save rack id for rotate on next M&D
           END_IF;
       END_IF;

   END_REGION

   REGION 3: Discharge
       // Open discharge solenoid and rack's return solenoid
       // Wait for discharge time
       // Close solenoids and release lock
       // Return to Off mode

       #TON_Discharge(IN := (#Status.iState = #eRoomMode_Discharge),
                      PT := #arrInFertigationSettings[#Status.iActiveRack].tDischargeTime);

       IF #Status.iState = #eRoomMode_Discharge THEN

           IF #TON_Discharge.Q OR #arrInFertigationSettings[#Status.iActiveRack].bEndDischargeCommand THEN
               #bEndDischarge := 1;
           END_IF;


           IF #bEndDischarge THEN
               #arrOutMutexLocks[#Status.iActiveRack] := #eRoomMode_Off;

               // wait until pump stops to close valves
               IF #arrInFertigationSettings[#Status.iActiveRack].bPumpAtStandstill THEN
                   #bDischargeSolenoidCommand := 0;
                   #arrOutReturnSolenoids[#Status.iActiveRack] := 0;
                   #Status.iLastMDRack := 0; // no rotate if last rack was discharged
                   #Status.iState := #eRoomMode_Off;
                   #bEndDischarge := 0;

               END_IF;

           ELSE
               #bDischargeSolenoidCommand := 1;
               #arrOutReturnSolenoids[#Status.iActiveRack] := 1;

           END_IF;

       END_IF;

   END_REGION

   REGION Nutrient Tank Mixing
       // 0: forced off, 1: forced on, 2: 10 minutes per day at noon, 3: Run for 24 hours then jump to mode 2

       #TON_24HourNutrientMix(IN := (#Controls.iNutrientMixingMode = #eNutrientMixingMode_FullDay),
                              PT := T#24h);

       IF #Controls.iNutrientMixingMode = #eNutrientMixingMode_Off THEN
           #bNutrientMixingCommand := 0;

       ELSIF #Controls.iNutrientMixingMode = #eNutrientMixingMode_On THEN
           #bNutrientMixingCommand := 1;

       ELSIF #Controls.iNutrientMixingMode = #eNutrientMixingMode_TenMinute THEN
           // Extract current PLC time
           #retVal := RD_LOC_T(OUT => #tCurrentDateTime);
           #tCurrentTime := DT_TO_TOD(IN := #tCurrentDateTime);

           IF (#tCurrentTime < #MIX_END_TIME) AND (#tCurrentTime > #MIX_START_TIME) THEN
               #bNutrientMixingCommand := 1;
           ELSE
               #bNutrientMixingCommand := 0;
           END_IF;

       ELSIF #Controls.iNutrientMixingMode = #eNutrientMixingMode_FullDay THEN

           IF #TON_24HourNutrientMix.Q THEN
               #bNutrientMixingCommand := 0;
               #Controls.iNutrientMixingMode := #eNutrientMixingMode_TenMinute;
           ELSE
               #bNutrientMixingCommand := 1;
           END_IF;

           // Catchall for incorrectly entered state, just turn off mixer
       ELSE
           #bNutrientMixingCommand := 0;
       END_IF;

   END_REGION

   REGION Set digital outputs
       #bOutTankReturnSolenoid := #bTankReturnSolenoidCommand;
       #bOutMPathSolenoid      := #bMPathSolenoidCommand;
       #bOutFreshWaterSolenoid := #bFreshWaterSolenoidCommand;
       #bOutDischargeSolenoid  := #bDischargeSolenoidCommand;
       #bOutNutrientMixing     := #bNutrientMixingCommand;
       #bOutNutrientA          := #bNutrientACommand;
       #bOutNutrientB          := #bNutrientBCommand;
       #bOutNutrientAcid       := #bNutrientAcidCommand;

   END_REGION
END_FUNCTION_BLOCK

FUNCTION_BLOCK "fbRoomMeasurementDosing"   // FB9, SCL
{ S7_Optimized_Access := 'TRUE' }
VERSION : 0.1
   VAR_INPUT
      bInStart : Bool;   // Start command for sequence
      iInActiveRack : Int;   // Current rack requesting MD
      iInPreviousRack : Int;   // Previous rack, if last operation was also MD (0 otherwise)
      rInTankLevel : Real;   // Current tank level (L)
      rInISEReading : Real;   // Current ISE sensor level
      rInECReading : Real;   // Current EC sensor level
      rInpHReading : Real;   // Current pH sensor level
      rInORPReading : Real;
      rInRackLevel : Real;   // Current rack reservoir level
      rInFreshLevelForMLoop : Real;
      rInFillLevelToPreviousShelf : Real;
      rInReturnPathVolume : Real;   // Return path volume (L) to fill from active rack
      rInTankEmptyLevel : Real;   // Volume at which tank is considered empty (L)
      InFertigationSettings : "udtFertigationSettings";   // Current rack fertigation settings
   END_VAR
   VAR_OUTPUT
      bOutTankReturnSolenoidCommand : Bool;   // Output for writing to tank return solenoid
      bOutActiveRackReturnSolenoidCommand : Bool;
      bOutActiveRackSupplySolenoidCommand : Bool;
      bOutPreviousRackReturnSolenoidCommand : Bool;
      bOutPreviousRackSupplySolenoidCommand : Bool;
      bOutFreshWaterSolenoidCommand : Bool;
      bOutDischargeSolenoidCommand : Bool;
      bOutMPathSolenoidCommand : Bool;
      bOutNutrientACommand : Bool;   // Output for writing to Nutrient A enable
      bOutNutrientBCommand : Bool;   // Output for writing to Nutrient B enable
      OutNutrientReadings : "udtNutrientReading";   // Final measured sensor levels for rack
      bOutDone : Bool;
   END_VAR
   VAR
      iState : Int;
      iNextState : Int;
      rTankStartingLevel : Real;
      TON_MeasurementTimer : TON_TIME;
      TON_NutrientATimer : TON_TIME;
      TON_NutrientBTimer : TON_TIME;
   END_VAR
   VAR CONSTANT
      eMDState_Idle : Int;
      eMDState_Rotate_Start : Int := 100;
      eMDState_Rotate_FillTankFromRack : Int := 102;
      eMDState_Rotate_PushToPrevious : Int := 104;
      eMDState_Rotate_FillTankFresh : Int := 106;
      eMDState_Rotate_MeasurementLoop : Int := 108;
      eMDState_Rotate_Done : Int := 119;
      eMDState_Measure_Start : Int := 120;
      eMDState_Measure_FillTankFromRack : Int := 122;
      eMDState_Measure_OpenMLoop : Int := 124;
      eMDState_Measure_Done : Int := 139;
      eMDState_Dosing_Start : Int := 140;
      eMDState_Dosing_AddNutrientA : Int := 142;
      eMDState_Dosing_AddNutrientB : Int := 144;
      eMDState_Dosing_AddFreshWater : Int := 146;
      eMDState_Dosing_Done : Int := 159;
      eMDState_Return_Start : Int := 160;
      eMDState_Return_FillPreviousRack : Int := 162;
      eMDState_Return_FillActiveRack : Int := 164;
      eMDState_Return_CloseSupplyPath : Int := 166;
      eMDState_Return_Done : Int := 169;
      iISEMode_Off : Int := 0;
      iISEMode_Load : Int := 1;
      iISEMode_Deplete : Int := 2;
   END_VAR
BEGIN
   REGION State 0: Idle
       // Wait for start command to move on to rotate if a previous rack used the piping 
       //  or directly to measure if not 

       IF #iState = #eMDState_Idle THEN
           #bOutDone := 0;
           IF #bInStart THEN
               IF #iInPreviousRack = 0 OR #iInPreviousRack = #iInActiveRack THEN
                   #iNextState := #eMDState_Measure_Start;
               ELSE
                   #iNextState := #eMDState_Rotate_Start;
               END_IF;
           END_IF;
       END_IF;


   END_REGION

   REGION State 100: Rotate
       // Open the tank return solenoid
       // Open the return solenoid and close the shelf solenoid for the current rack until a fixed amount of water is pumped into the tank
       // Close the return solenoid of the current rack and open the supply valve of the previous rack to push 19L from the 
       //     tank into the previous rack. 
       //     

       // Open tank return and rack return, close shelf, record starting tank level, then move to next state
       IF #iState = #eMDState_Rotate_Start THEN
           #bOutTankReturnSolenoidCommand := 1; 
           #bOutActiveRackReturnSolenoidCommand := 1;
           #iNextState := #eMDState_Rotate_FillTankFromRack;
           #rTankStartingLevel := #rInTankLevel;
       END_IF;

       // Once the target fill level is reached, close the return solenoids, open the previous rack's supply, then move to next state
       IF #iState = #eMDState_Rotate_FillTankFromRack THEN
           IF #rInTankLevel >= #rTankStartingLevel + #rInReturnPathVolume THEN
               #bOutActiveRackReturnSolenoidCommand := 0;
               #bOutPreviousRackSupplySolenoidCommand := 1;
               #bOutTankReturnSolenoidCommand := 1;
               #iNextState := #eMDState_Rotate_PushToPrevious;
           END_IF;
       END_IF;

       // Run until 19L have been pushed into the previous rack and the tank is back at its original level, then close the
       // previous rack's supply solenoid and move to next state
       IF #iState = #eMDState_Rotate_PushToPrevious THEN

           IF #rInTankLevel <= #rTankStartingLevel THEN
               #bOutPreviousRackSupplySolenoidCommand := 0;
               #iNextState := #eMDState_Rotate_FillTankFresh;
           END_IF;

       END_IF;

       // Open the fresh water supply and fill the tank until the target level is reached, then close the fresh water supply, open the
       // measurement path solenoid and the discharge solenoid and move to the next state
       IF #iState = #eMDState_Rotate_FillTankFresh THEN

           IF #rInTankLevel >= #rTankStartingLevel + #rInFreshLevelForMLoop THEN
               #bOutFreshWaterSolenoidCommand := 0;
               #bOutMPathSolenoidCommand := 1;
               #bOutDischargeSolenoidCommand := 1;
               #iNextState := #eMDState_Rotate_MeasurementLoop;
           ELSE
               #bOutFreshWaterSolenoidCommand := 1;
           END_IF;
       END_IF;

       // Push water out through the measurement loop. Once the tank is empty, close measurement path solenoid and
       // the discharge solenoid and move to the next state
       IF #iState = #eMDState_Rotate_MeasurementLoop THEN

           IF #rInTankLevel <= #rInTankEmptyLevel THEN

               #bOutMPathSolenoidCommand := 0;
               #bOutDischargeSolenoidCommand := 0;
               #iNextState := #eMDState_Rotate_Done;
           END_IF;
       END_IF;

       IF #iState = #eMDState_Rotate_Done THEN
           #iNextState := #eMDState_Measure_Start;
       END_IF;

   END_REGION

   REGION State 120: Measure
       // Receive water from rack and start measurement phase. Open measurement loop, push water through, record sensor readings, 
       // determine setpoints, and move on to dosing

       #TON_MeasurementTimer(IN := (#iState = #eMDState_Measure_OpenMLoop),
                            PT := #InFertigationSettings.tMeasurementTime);

       // Open tank return and shelf return solenoid
       IF #iState = #eMDState_Measure_Start THEN
           #bOutTankReturnSolenoidCommand := 1;
           #bOutActiveRackReturnSolenoidCommand := 1;
           #iNextState := #eMDState_Measure_FillTankFromRack;
           #rTankStartingLevel := #rInTankLevel;
       END_IF;

       // Wait to receive target level from rack, close rack return solenoid
       IF #iState = #eMDState_Measure_FillTankFromRack THEN
           IF #rInTankLevel >= #InFertigationSettings.rMeasurementVolume THEN
               #iNextState := #eMDState_Measure_OpenMLoop;
               #bOutActiveRackReturnSolenoidCommand := 0;
           END_IF;
       END_IF;

       // Open MPath solenoid, wait for measurement time then record measurement
       IF #iState = #eMDState_Measure_OpenMLoop THEN

           IF #TON_MeasurementTimer.Q THEN
               #OutNutrientReadings.rISEReading := #rInISEReading;
               #OutNutrientReadings.rECReading := #rInECReading;
               #OutNutrientReadings.rpHReading := #rInpHReading;
               #OutNutrientReadings.rORPReading := #rInORPReading;
               #bOutMPathSolenoidCommand := 0;
               #bOutTankReturnSolenoidCommand := 0;
               #iNextState := #eMDState_Measure_Done;
           ELSE
               #bOutMPathSolenoidCommand := 1;
           END_IF;
       END_IF;


       IF #iState = #eMDState_Measure_Done THEN
           #iNextState := #eMDState_Dosing_Start;
       END_IF;


   END_REGION

   REGION State 140: Dosing

       // Check if rack fertigation logic has requested dosing
       // Add enabled nutrients one at a time for dosing time then add fresh water to tank

       IF #iState = #eMDState_Dosing_Start THEN

           IF #InFertigationSettings.bDosingActive THEN

               IF #InFertigationSettings.bNutrientAEnable THEN
                   #iNextState := #eMDState_Dosing_AddNutrientA;
               ELSIF #InFertigationSettings.bNutrientBEnable THEN
                   #iNextState := #eMDState_Dosing_AddNutrientB;
               ELSE
                   #iNextState := #eMDState_Dosing_Done;
               END_IF;

           ELSE
               #iNextState := #eMDState_Dosing_Done;
           END_IF;
       END_IF;

       #TON_NutrientATimer(IN := (#iState = #eMDState_Dosing_AddNutrientA),
                          PT := #InFertigationSettings.tNutrientDosingDuration);
       // Add nutrient A for dosing time, then check if nutrient B is needed
       IF #iState = #eMDState_Dosing_AddNutrientA THEN

           IF #TON_NutrientATimer.Q THEN
               #bOutNutrientACommand := 0;
               IF #InFertigationSettings.bNutrientBEnable THEN
                   #iNextState := #eMDState_Dosing_AddNutrientB;
               ELSE
                   #iNextState := #eMDState_Dosing_AddFreshWater;
               END_IF;
           ELSE
               #bOutNutrientACommand := 1;
           END_IF;
       END_IF;

       #TON_NutrientBTimer(IN := (#iState = #eMDState_Dosing_AddNutrientB),
                          PT := #InFertigationSettings.tNutrientDosingDuration);
       // Add nutrient B for dosing time, then move on to water fill
       IF #iState = #eMDState_Dosing_AddNutrientB THEN

           IF #TON_NutrientBTimer.Q THEN
               #bOutNutrientBCommand := 0;
               #iNextState := #eMDState_Dosing_AddFreshWater;
           ELSE
               #bOutNutrientBCommand := 1;
           END_IF;
       END_IF;

       // Add fresh water to tank if tank level plus rack is less than the operating volume
       IF #iState = #eMDState_Dosing_AddFreshWater THEN
           IF ((#rInTankLevel + #rInRackLevel) < #InFertigationSettings.rOperatingVolume) THEN
               #bOutFreshWaterSolenoidCommand := 1;
           ELSE
               #bOutFreshWaterSolenoidCommand := 0;
               #iNextState := #eMDState_Dosing_Done;
           END_IF;
       END_IF;


       IF #iState = #eMDState_Dosing_Done THEN
           #iNextState := #eMDState_Return_Start;
       END_IF;

   END_REGION

   REGION State 160: Return TO Tank
       // If a previous rack was used, open supply path to previous rack, wait for 8L drop in tank
       // Open supply path to active rack, activate floor pump, wait for tank contents to return to rack
       // Close supply path

       // Determine which rack to start return to
       IF #iState = #eMDState_Return_Start THEN

           IF #iInPreviousRack = 0 OR #iInPreviousRack = #iInActiveRack  THEN
               #iNextState := #eMDState_Return_FillActiveRack;
           ELSE
               #iNextState := #eMDState_Return_FillPreviousRack;
           END_IF;
           #rTankStartingLevel := #rInTankLevel;
       END_IF;

       // Open supply path to previous rack, wait for 8L drop in tank, close previous rack return path
       IF #iState = #eMDState_Return_FillPreviousRack THEN
           #bOutPreviousRackSupplySolenoidCommand := 1;
           IF #rInTankLevel < (#rTankStartingLevel - #rInFillLevelToPreviousShelf) THEN
               #bOutPreviousRackSupplySolenoidCommand := 0;
               #iNextState := #eMDState_Return_FillActiveRack;
           END_IF;
       END_IF;

       // Open supply path to active rack
       IF #iState = #eMDState_Return_FillActiveRack THEN
           #rTankStartingLevel := #rInTankLevel;
           #bOutActiveRackSupplySolenoidCommand := 1;
           #iNextState := #eMDState_Return_CloseSupplyPath;
       END_IF;

       // Wait for tank to empty, close supply path
       IF #iState = #eMDState_Return_CloseSupplyPath THEN
           IF #rInTankLevel <= #rInTankEmptyLevel OR #rInRackLevel >= #InFertigationSettings.rMaxReservoirVolume THEN
               #bOutActiveRackSupplySolenoidCommand := 0;
               #iNextState := #eMDState_Return_Done;
           END_IF;
       END_IF;

       //Return to Idle at end of M&D
       IF #iState = #eMDState_Return_Done THEN
           #bOutDone := 1;
           #iNextState := #eMDState_Idle;
       END_IF;

   END_REGION


   REGION Update State
       IF #iState <> #iNextState THEN
           #iState := #iNextState;
       END_IF;
   END_REGION
END_FUNCTION_BLOCK

FUNCTION_BLOCK "fbRackPump"   // FB10, LAD
{ S7_Optimized_Access := 'TRUE' }
VERSION : 0.1
// Pump has 3 modes: Off, Priming, Running. 
// If the pump speed changes from zero to non-zero, start priming for the priming duration
// Once priming is complete, move to Pump running while the rack remains in Fill or Circulate
   VAR_INPUT
      rInSpeedCommand : Real;   // Commanded pump speed (%)
   END_VAR
   VAR RETAIN
      Controls : Struct
         rPrimeSpeed : Real := 100.0;   // Pump speed when priming (%)
         diPrimingSecs : DInt := 60;   // Duration of pump priming (seconds)
         bOverrideEnable : Bool;   // Sets pump speed to the override value
         rOverrideSpeed : Real;   // Manual override speed (%) Set to 0 to turn off.
      END_STRUCT;
   END_VAR
   VAR
      Status : Struct
         iState : Int;   // 0: Off, 1: Priming, 2:Running
         rCommandSpeed : Real;   // Speed commanded to VFD (%)
         rActualSpeed : Real;   // Speed reported from VFD (%)
         rVoltage : Real;   // Vrms
         rCurrent : Real;   // Arms
         rPower : Real;   // kW
         rPowerFactor : Real;
         bError : Bool;
         ErrorDetail : "udtError_VFD";
      END_STRUCT;
      fbVFD : "fbVFD_GSeries";
      TON_Priming : TON_TIME;
      dummyUdt : "udtHMI_VFD_Control";   // Ignore
   END_VAR
   VAR_TEMP
      arrTelegramWords : Array[1..6] of Int;
      iRet : Int;
   END_VAR
   VAR CONSTANT
      eStateOff : Int := 0;
      eStatePriming : Int := 1;
      eStateRunning : Int := 2;
      cScalingFactor : Real := 16384.0;   // Full scale (100%) value of VFD parameters
   END_VAR
BEGIN

REGION Network 1 (SCL): Determine pump VFD command speed based on off/priming/run state
   IF #rInSpeedCommand <> 0 THEN
       // start out by priming, then switch to running
       IF #Status.iState = #eStateOff THEN
           #Status.iState := #eStatePriming;
       ELSIF #Status.iState = #eStatePriming AND #TON_Priming.Q THEN
           #Status.iState := #eStateRunning;
       END_IF;

   ELSE
       #Status.iState := #eStateOff;
   END_IF;

   #TON_Priming(IN := (#Status.iState = #eStatePriming),
                PT := DINT_TO_TIME(#Controls.diPrimingSecs * 1000));

   // Check for manual override
   IF #Controls.bOverrideEnable THEN
       #fbVFD.rInCommandSpeed := #Controls.rOverrideSpeed;

   ELSE
       CASE #Status.iState OF
           #eStateOff: // Off
               #fbVFD.rInCommandSpeed := 0;
           #eStatePriming: // Priming - run at priming speed until priming timer has elapsed then transition to Running   
               #fbVFD.rInCommandSpeed := #Controls.rPrimeSpeed;
           #eStateRunning: // Running
               #fbVFD.rInCommandSpeed := #rInSpeedCommand;
       END_CASE;

       // if override is not active, override speed tracks command speed so that activating override mode
       // doesn't unexpectedly change the value
       #Controls.rOverrideSpeed := #fbVFD.rInCommandSpeed;

   END_IF;

   #Status.rCommandSpeed := #fbVFD.rInCommandSpeed;
END_REGION

REGION Network 2: Open library G series VFD block call
   // Telegram is assigned globally in fbConfig.
   // Contactor output is fed back since we con't have a physical one.
   // Dummy Udt is needed even though we don't have an HMI faceplate.
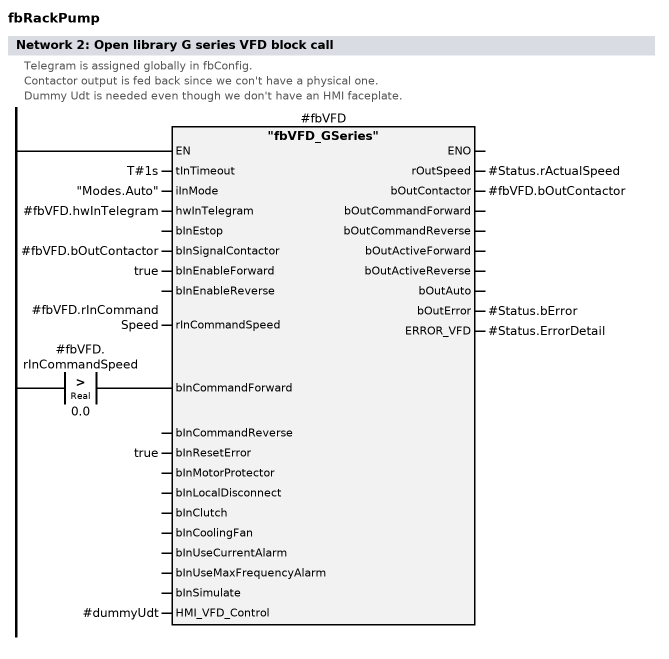
   RUNG wire#powerrail
      #fbVFD(bInCommandForward := wire#w1, tInTimeout := T#1s, iInMode := "Modes.Auto", hwInTelegram := #fbVFD.hwInTelegram, bInEstop :=, bInSignalContactor := #fbVFD.bOutContactor, bInEnableForward := true, bInEnableReverse :=, rInCommandSpeed := #fbVFD.rInCommandSpeed, bInCommandReverse :=, bInResetError := true, bInMotorProtector :=, bInLocalDisconnect :=, bInClutch :=, bInCoolingFan :=, bInUseCurrentAlarm :=, bInUseMaxFrequencyAlarm :=, bInSimulate :=, HMI_VFD_Control := #dummyUdt, rOutSpeed => #Status.rActualSpeed, bOutContactor => #fbVFD.bOutContactor, bOutCommandForward =>, bOutCommandReverse =>, bOutActiveForward =>, bOutActiveReverse =>, bOutAuto =>, bOutError => #Status.bError, ERROR_VFD => #Status.ErrorDetail)
   END_RUNG
   RUNG wire#powerrail
      { S7_Templates := "SrcType := Real" } GT_Contact(in1 := #fbVFD.rInCommandSpeed, in2 := 0.0)
   END_RUNG wire#w1
   // the same network as SCL:
   #fbVFD(tInTimeout := T#1s,   // "fbVFD_GSeries"
          iInMode := "Modes.Auto",
          hwInTelegram := #fbVFD.hwInTelegram,
          bInSignalContactor := #fbVFD.bOutContactor,
          bInEnableForward := true,
          rInCommandSpeed := #fbVFD.rInCommandSpeed,
          bInCommandForward := #fbVFD.rInCommandSpeed > 0.0,
          bInResetError := true,
          HMI_VFD_Control := #dummyUdt,
          rOutSpeed => #Status.rActualSpeed,
          bOutContactor => #fbVFD.bOutContactor,
          bOutError => #Status.bError,
          ERROR_VFD => #Status.ErrorDetail);
END_REGION

REGION Network 3 (SCL): Read additional drive parameters from exteneded telegram
   #iRet := DPRD_DAT(LADDR := #fbVFD.hwInTelegram, RECORD => #arrTelegramWords);

   // Telegram word 1 (status word) is handled inside fbVFD
   #Status.rActualSpeed := #arrTelegramWords[2] / #cScalingFactor * 100; // percent 
   #Status.rVoltage := #arrTelegramWords[3] / #cScalingFactor * 1000; // Vrms
   #Status.rCurrent := #arrTelegramWords[4] / #cScalingFactor * 5.8;//9.43; // Arms
   #Status.rPower := #arrTelegramWords[5] / #cScalingFactor * 1.49;//3.15; // Kw
   #Status.rPowerFactor := #arrTelegramWords[6] / #cScalingFactor;
END_REGION
END_FUNCTION_BLOCK

FUNCTION_BLOCK "fbConfig"   // FB11, SCL
{ S7_Optimized_Access := 'TRUE' }
VERSION : 0.1
   VAR_INPUT
      bInSimulation : Bool := false;   // If true, skips IO reconfig steps
   END_VAR
   VAR RETAIN
      Controls : Struct
         iSetNumRooms : Int := 1;
         arrSetNumRacksPerRoom : Array[1.."MAX_ROOMS"] of Int;
         bSetConfig : Bool := false;
      END_STRUCT;
   END_VAR
   VAR
      Status : Struct
         bDone : Bool;
         bBusy : Bool;
         bError : Bool;
         ErrorMsg : String;
      END_STRUCT;
      iNumRooms : Int := 0;
      iStep : Int;
      iNextStep : Int;
      R_TRIG_SetConfig : R_TRIG;
      ReconfigIOSystem : ReconfigIOSystem;
      arrVfdDeviceConfig : Array[-2.."MAX_VFDS"] of Word;
   END_VAR
   VAR_TEMP
      iRoomIndex : Int;
      iRackIndex : Int;
      arrTelegrams : Array[1.."MAX_VFDS"] of HW_SUBMODULE;
      arrIoDeviceIds : Array[1.."MAX_VFDS"] of HW_DEVICE;
      i : Int;
      iVfdCount : Int;
      bSettingsValid : Bool;
      strErrorCode : String;
      retVal : Word;
   END_VAR
   VAR CONSTANT
      eStep_ValidateConfig : Int;
      eStep_SetUp : Int := 1;
      eStep_Deactivate : Int := 2;
      eStep_WaitForDeactivate : Int := 3;
      eStep_Reconfig : Int := 4;
      eStep_WaitForReconfig : Int := 5;
      eStep_Restart : Int := 6;
      eStep_Done : Int := 7;
      eStep_Error : Int := 8;
   END_VAR
   // Controls.arrSetNumRacksPerRoom[1] := 6;
BEGIN
   // Enables VFDs and IO racks based on the number of configured rooms and racks.
   // The intention is for everything to be configurable via the OPC UA interface and nothing
   // needs to be changed in TIA Portal, so that all deployments regardless of size can use the same codebase.

   // Global constants for reference:
   (*
   "MAX_ROOMS"
   "MAX_RACKS_PER_ROOM"
   "MAX_VFDS"

   "NUM_AI_ROOM"
   "NUM_AI_RACK"
   "MAX_AI_TOTAL"

   "NUM_DQ_ROOM"
   "NUM_DQ_RACK"
   "MAX_DQ_TOTAL"
   *)

   REGION 0: Validate config, set num racks and rooms

       // wait for start command
       #R_TRIG_SetConfig(CLK:= #Controls.bSetConfig);

       // also trigger on PLC startup
       IF "FirstScan" OR #iStep = #eStep_ValidateConfig OR
           (#R_TRIG_SetConfig.Q AND (#iStep = #eStep_Done OR #iStep = #eStep_Error) ) THEN

           REGION Check error conditions            
               // make sure specified number of rooms and racks is valid
               #bSettingsValid := TRUE;
               #Status.ErrorMsg := '';

